(* CODESYS project BatteryPicker.project
   Company: LCP
   DefaultNamespace: LCP_RoboticApplication
   Title: LCP_PnP_Motion_Master
   Version: 1.0

Project tree, tasks and I/O mapping:
  Controller_3200C : Controller 3200C, Lenze, order no. LPC 1000, version 3.13.0.2
    application Application
      libraries: ModbusTCP Slave, * (3S - Smart Software Solutions GmbH); CAA Types, 3.0.0.2 (3S - Smart Software Solutions GmbH); CAA File, * (CAA Technical Workgroup); L_CT1P_ControlToolbox, * (Lenze); L_Util, 3.13.0.0 (Lenze); L_PLCDataManagerAccess, 3.0.0.0 (Lenze); L_PLCLoggingAccess, 3.3.0.0 (Lenze); L_IE1P_ApplicationErrors, 3.13.1.0 (Lenze); L_MC4P_RoboticHandling, 3.13.2.5 (Lenze); L_IODrvEtherCAT, 3.12.0.0 (Lenze); SysTimeCore, * (System); CAA Net Base Services, * (CAA Technical Workgroup); L_USPP_SignalProcessing, * (Lenze); L_MC1P_MotionControlBasic, 3.13.1.0 (Lenze); L_MC2P_MotionControlCam, 3.13.1.56 (Lenze); L_DCO_DriveCommunication, 3.1.0.0 (Lenze); SysMem, * (System); CAA Mathematics, * (CAA Technical Workgroup); LCP_PnP_Ellipse_Motion, 2.0 (LCP); CAA Memory, * (CAA Technical Workgroup)
      task Motion (cyclic, interval t#1ms, priority 1, watchdog t#2ms x 1) calls Main
      task Logic (cyclic, interval t#5ms, priority 2) calls LogicControl
      program Main [ST]: A00_Init, A20_ManualJog, A30_AutoRun, A80_SuckBlow, A60_CameraHandler, A93_SetTorqueLimit, A02_DetectDeviceChoose, A03_PowerCtrl, A04_ResetFunction, A40_SetParameters, A94_RealAxisFilter, A96_IK, A98_TFFControl
      B0_GloabalVariables/
        global variables PersistentVars
        global variables L_MC4P_AGBC_VARS
        global variables GVL_Const
        global variables PrgVars
        global variables GVL_MainFlow
        global variables PPVars
        global variables GVL_HardwareIO
      B1_STRUCT/
        data type sRobotPos
        data type CalibratePt
        data type Detect_Device
        data type Display_Product
      B5_VISUAL/
        visualisation DeltaRobot
        visualisation ABControl
        visualisation Products
        visualisation SensorBuffer
        visualisation MultiPick
      program LogicControl [ST]: A40_Modbus_Slave, A20_StatusDisplay, A10_CameraInterface, A01_EditPrg, A10_Homing, A50_Brake
      B6_TRACE/
        trace RobotStatus (task Motion): CustomerPrgHandling.iAutoStep, Delta_Robot.lrPathVelocity, Delta_Robot.lrPathAcceleration, CustomerPrgHandling.BoxBuffer.NewProd_Rtrig.Q, Infeeder.lrActPosition, Infeeder.lrActVelocity, Infeeder.lrActAcceleration, CustomerPrgHandling.MC_TrackConveyorBelt_U1.Busy, CustomerPrgHandling.MC_TrackConveyorBelt_U1.Active, CustomerPrgHandling.MC_TrackConveyorBelt_U1.InSync, CustomerPrgHandling.MC_TrackConveyorBelt_U1.Done, Outfeeder.lrActPosition, Outfeeder.lrActVelocity, Outfeeder.lrActAcceleration, CustomerPrgHandling.MC_TrackConveyorBelt_U2.Busy, CustomerPrgHandling.MC_TrackConveyorBelt_U2.Active, CustomerPrgHandling.MC_TrackConveyorBelt_U2.InSync, CustomerPrgHandling.MC_TrackConveyorBelt_U2.Done, CustomerPrgHandling.MC_TrackConveyorBelt_U2.Abort, CustomerPrgHandling.MC_TrackConveyorBelt_U2.CommandAborted, CustomerPrgHandling.L_RPP_PickPlace_0.Busy, CustomerPrgHandling.L_RPP_PickPlace_1.Busy, CustomerPrgHandling.L_RPP_PickPlace_1.xBusyTemp, CustomerPrgHandling.L_RPP_PickPlace_1.SWOut, CustomerPrgHandling.MoveToWaitPoint0.Busy, CustomerPrgHandling.MoveToWaitPoint0.Active, CustomerPrgHandling.MoveToWaitPoint0.Done, CustomerPrgHandling.BoxBuffer.xFirstProdDel, CustomerPrgHandling.BoxBuffer.xProdInfoReady, CustomerPrgHandling.BoxBuffer.sFirstProdInfo.lrDeltaX, CustomerPrgHandling.BoxBuffer.lrPosFirstProdInfo, CustomerPrgHandling.BoxBuffer.iNewProdCount, A1.lrActTorque, A2.lrActTorque, A3.lrActTorque, AxisYaw.lrActTorque, A1.lrActFollowingError, A2.lrActFollowingError, A3.lrActFollowingError, AxisYaw.lrActFollowingError
        trace Trace (task Motion): Axis_X.lrSetPosition, Axis_Y.lrSetPosition, Axis_Z.lrSetPosition, Axis_X.lrActPosition, Axis_Y.lrActPosition, Axis_Z.lrActPosition, Axis_X.lrSetAcceleration, Axis_Y.lrSetAcceleration, Axis_Z.lrSetAcceleration, Delta_Robot.lrPathVelocity, Delta_Robot.lrPathAcceleration, A1.lrSetAcceleration, A2.lrSetAcceleration, A3.lrSetAcceleration, A1.lrActPosition, A2.lrActPosition, A3.lrActPosition, A1.lrActTorque, A2.lrActTorque, A3.lrActTorque, A1.lrActFollowingError, A2.lrActFollowingError, A3.lrActFollowingError
        trace RobotPerformance (task Motion): CustomerPrgHandling.L_RPP_PickPlace_0.Busy, CustomerPrgHandling.L_RPP_PickPlace_1.Busy, Axis_X.lrSetPosition, Axis_Y.lrSetPosition, Axis_Z.lrSetPosition, Axis_X.lrActPosition, Axis_Y.lrActPosition, Axis_Z.lrActPosition, Axis_X.lrSetAcceleration, Axis_Y.lrSetAcceleration, Axis_Z.lrSetAcceleration, Delta_Robot.lrPathVelocity, Delta_Robot.lrPathAcceleration, A1.lrActPosition, A2.lrActPosition, A3.lrActPosition, A1.lrActTorque, A2.lrActTorque, A3.lrActTorque, A1.lrActFollowingError, A2.lrActFollowingError, A3.lrActFollowingError
        trace ErrorID (task Motion): DeltaRobot_ErrorID, A1axis_ErrorID, A2axis_ErrorID, A3axis_ErrorID, AuxCaxis_ErrorID, Xaxis_ErrorID, Yaxis_ErrorID, Zaxis_ErrorID, ErrorID, Main.LoadDistribution.xOverlap, Main.LoadDistribution.xProductNew
        trace Trace_1 (task Motion): CustomerPrgHandling.iAutoStep
        trace PathLength_DurationInternal (task Motion): CustomerPrgHandling.L_RPP_PickPlace_0.Ellipse_Cal_Pts.lrPathLength, CustomerPrgHandling.L_RPP_PickPlace_1.Ellipse_Cal_Pts.lrPathLength, CustomerPrgHandling.L_RPP_PickPlace_0.lrDurationInternal, CustomerPrgHandling.L_RPP_PickPlace_1.lrDurationInternal
        trace Trace_2 (task Motion): CustomerPrgHandling.L_RPP_PickPlace_0.Busy, CustomerPrgHandling.L_RPP_PickPlace_1.Busy, Axis_X.lrSetPosition, Axis_Y.lrSetPosition, Axis_Z.lrSetPosition, Axis_X.lrActPosition, Axis_Y.lrActPosition, Axis_Z.lrActPosition, Axis_X.lrSetAcceleration, Axis_Y.lrSetAcceleration, Axis_Z.lrSetAcceleration, Delta_Robot.lrPathVelocity, Delta_Robot.lrPathAcceleration, A1.lrActPosition, A2.lrActPosition, A3.lrActPosition, A1.lrActTorque, A2.lrActTorque, A3.lrActTorque, A1.lrActFollowingError, A2.lrActFollowingError, A3.lrActFollowingError
      program CustomerPrgHandling [ST]: A01_PickAlone, A02_PlaceAlone, A00_ProgramHandling, A03_RobotSateTransition
      FunctionBlock/
        function block FourPts_Calibration [ST]
        function _L_MC1B_PackBytesToDWord [ST]
        function _L_MC1B_PackBytesToLreal [ST]
        function _L_MC1B_PackBytesToWord [ST]
        function _L_MC1B_PackDWordToByte [ST]
        function _L_MC1B_PackLRealToByte [ST]
        function _L_MC1B_PackWordToByte [ST]
      TorqueFeedforwardControl/
        trace Dynamics (task TaskHighPriority): Axis_X.lrSetPosition, Axis_Y.lrSetPosition, Axis_Z.lrSetPosition, Axis_X.lrSetVelocity, Axis_Y.lrSetVelocity, Axis_Z.lrSetVelocity, Axis_X.lrSetAcceleration, Axis_Y.lrSetAcceleration, Axis_Z.lrSetAcceleration, A1.lrSetPosition, A2.lrSetPosition, A3.lrSetPosition, A1.lrSetVelocity, A2.lrSetVelocity, A3.lrSetVelocity, A1.lrSetAcceleration, A2.lrSetAcceleration, A3.lrSetAcceleration, A1.lrActTorque, A2.lrActTorque, A3.lrActTorque, A1.lrActFollowingError, A2.lrActFollowingError, A3.lrActFollowingError
        trace Trace_Theta (task Motion): Main.fb_InverseKinematics.theta1, Main.fb_InverseKinematics.theta2, Main.fb_InverseKinematics.theta3, A1.lrSetPosition, A2.lrSetPosition, A3.lrSetPosition
        trace Trace_Torque (task Motion): CustomerPrgHandling.L_RPP_PickPlace_1.Busy, A1.lrActTorque, A2.lrActTorque, A3.lrActTorque, Axis_X.lrSetPosition, Axis_Y.lrSetPosition, Axis_Z.lrSetPosition, Main.LCP_MC4P_TorqueComputation_1.alrComputedTorque[1], Main.LCP_MC4P_TorqueComputation_1.alrComputedTorque[2], Main.LCP_MC4P_TorqueComputation_1.alrComputedTorque[3], Main.LCP_MC4P_TorqueComputation_1.alrSetTorqueOut[1], Main.LCP_MC4P_TorqueComputation_1.alrSetTorqueOut[2], Main.LCP_MC4P_TorqueComputation_1.alrSetTorqueOut[3], A1.lrSetTorqueToDrive, A2.lrSetTorqueToDrive, A3.lrSetTorqueToDrive, A1.lrActFollowingError, A2.lrActFollowingError, A3.lrActFollowingError
        trace Torque (task Motion): A1.lrActTorque, A2.lrActTorque, A3.lrActTorque, Main.fb_SimplifiedTorqueComputationKorea.tau1, Main.fb_SimplifiedTorqueComputationKorea.tau2, Main.fb_SimplifiedTorqueComputationKorea.tau3, Main.fb_SimplifiedTorqueComputationGermany.tau1, Main.fb_SimplifiedTorqueComputationGermany.tau2, Main.fb_SimplifiedTorqueComputationGermany.tau3, Main.fb_CompleteTorqueComputationSpain.tau1, Main.fb_CompleteTorqueComputationSpain.tau2, Main.fb_CompleteTorqueComputationSpain.tau3, Main.lrAverageTorque[1], Main.lrAverageTorque[2], Main.lrAverageTorque[3], A1.lrActFollowingError, A2.lrActFollowingError, A3.lrActFollowingError, A1.lrSetTorqueToDrive, A2.lrSetTorqueToDrive, A3.lrSetTorqueToDrive
        trace Trace_4 (task Motion): CustomerPrgHandling.L_RPP_PickPlace_0.Busy, A1.lrActTorque, A2.lrActTorque, A3.lrActTorque, Main.fb_SimplifiedTorqueComputation.tau1, Main.fb_SimplifiedTorqueComputation.tau2, Main.fb_SimplifiedTorqueComputation.tau3, Main.fb_SimplifiedTorqueComputation.alrFriction[1], Main.fb_SimplifiedTorqueComputation.alrFriction[2], Main.fb_SimplifiedTorqueComputation.alrFriction[3], A1.lrSetTorqueToDrive, A2.lrSetTorqueToDrive, A3.lrSetTorqueToDrive, A1.lrActFollowingError, A2.lrActFollowingError, A3.lrActFollowingError
        trace Torque_1 (task Motion): CustomerPrgHandling.L_RPP_PickPlace_0.Busy, A1.lrActTorque, A2.lrActTorque, A3.lrActTorque, Main.fb_SimplifiedTorqueComputationGermany.tau1, Main.fb_SimplifiedTorqueComputationGermany.tau2, Main.fb_SimplifiedTorqueComputationGermany.tau3, Main.fb_SimplifiedTorqueComputationGermany.alrFriction[1], Main.fb_SimplifiedTorqueComputationGermany.alrFriction[2], Main.fb_SimplifiedTorqueComputationGermany.alrFriction[3], A1.lrActFollowingError, A2.lrActFollowingError, A3.lrActFollowingError, A1.lrSetTorqueToDrive, A2.lrSetTorqueToDrive, A3.lrSetTorqueToDrive
        trace Trace_5 (task Motion): Main.fb_InverseKinematics.theta1, Main.fb_InverseKinematics.theta2, Main.fb_InverseKinematics.theta3, A1.lrSetPosition, A2.lrSetPosition, A3.lrSetPosition
        trace Trace_6 (task Motion): A1.lrActTorque, A2.lrActTorque, A3.lrActTorque, Main.fb_SimplifiedTorqueComputationKorea.tau1, Main.fb_SimplifiedTorqueComputationKorea.tau2, Main.fb_SimplifiedTorqueComputationKorea.tau3, Main.fb_SimplifiedTorqueComputationGermany.tau1, Main.fb_SimplifiedTorqueComputationGermany.tau2, Main.fb_SimplifiedTorqueComputationGermany.tau3, Main.fb_CompleteTorqueComputationSpain.tau1, Main.fb_CompleteTorqueComputationSpain.tau2, Main.fb_CompleteTorqueComputationSpain.tau3, Main.lrAverageTorque[1], Main.lrAverageTorque[2], Main.lrAverageTorque[3], A1.lrActFollowingError, A2.lrActFollowingError, A3.lrActFollowingError, A1.lrSetTorqueToDrive, A2.lrSetTorqueToDrive, A3.lrSetTorqueToDrive
        trace L_TT1P_TrackPickAndPlace (task TaskHighPriority): Axis_X.lrSetPosition, Axis_Y.lrSetPosition, Axis_Z.lrSetPosition, Axis_X.lrSetVelocity, Axis_Y.lrSetVelocity, Axis_Z.lrSetVelocity, Axis_X.lrSetAcceleration, Axis_Y.lrSetAcceleration, Axis_Z.lrSetAcceleration, A1.lrSetPosition, A2.lrSetPosition, A3.lrSetPosition, A1.lrSetVelocity, A2.lrSetVelocity, A3.lrSetVelocity, A1.lrSetAcceleration, A2.lrSetAcceleration, A3.lrSetAcceleration, A1.lrActTorque, A2.lrActTorque, A3.lrActTorque, A1.lrActFollowingError, A2.lrActFollowingError, A3.lrActFollowingError
        trace LCP_MC4P_MoveBSpline (task Motion): Axis_X.lrSetPosition, Axis_Y.lrSetPosition, Axis_Z.lrSetPosition, Axis_X.lrSetVelocity, Axis_Y.lrSetVelocity, Axis_Z.lrSetVelocity, Axis_X.lrSetAcceleration, Axis_Y.lrSetAcceleration, Axis_Z.lrSetAcceleration, A1.lrSetPosition, A2.lrSetPosition, A3.lrSetPosition, A1.lrSetVelocity, A2.lrSetVelocity, A3.lrSetVelocity, A1.lrSetAcceleration, A2.lrSetAcceleration, A3.lrSetAcceleration, A1.lrActTorque, A2.lrActTorque, A3.lrActTorque, A1.lrActFollowingError, A2.lrActFollowingError, A3.lrActFollowingError
        trace ErrorAnalysis (task ): xSystemWarning, xSystemError, ErrorID, WarningID, Delta_Robot.eActiveErrorID, Axis_X.eActiveErrorID, Axis_Y.eActiveErrorID, Axis_Z.eActiveErrorID, A1.eActiveErrorID, A2.eActiveErrorID, A3.eActiveErrorID
      A10-Structs/
        A11-scCommunication/
          data type scDataMotion_FromPLC
          data type scDataMotion_ToPLC
        A12_scControlWord/
          data type scDataControlWord_1_FromPLC
        A13_scStatusWord/
          data type scDataMotionStatusWord_1_ToPLC
        A14_scPnP_Data/
          data type scPnP_Data
        data type scWord_to_bits
        A15_SlaveStatetoMaster/
          data type eSlaveToMaster_State
      A20-Unions/
        data type scDataMotion_ToSiemens
        data type scDataMotion_FromSiemens
      A30_Enum/
        A31_AutoRunStep/
          data type eAutoRun_Step
    Coupler_I_O_moduls : Coupler I/O moduls, Lenze, version 3.6.0.0
        settings: Count groups = 1; Application Name of Task = 'Application'; Group1 Task Name = 'Motion'
        unmapped channels: Error, unused, unused, unused, unused, unused, unused, unused, ErrorID, AbsoluteCounter, ErrorReset, unused, unused, unused, unused, unused, unused, unused
      EPM_S202 : EPM-S202: DI8, DC 24V, Lenze, order no. EPM-S202, version 3.6.0.0
          settings: Group = 0; Task Guid = '00000000-0000-0000-0000-000000000000'
          unmapped channels: DI1, DI2, DI3, DI4, DI5, DI6, DI7, DI8
      EPM_S302 : EPM-S302: DO8, DC 24V, 0.5A, Lenze, order no. EPM-S302, version 3.6.0.0
          settings: Group = 0; Task Guid = '00000000-0000-0000-0000-000000000000'
          unmapped channels: DO1, DO2, DO3, DO4, DO5, DO6, DO7, DO8
    AxesGroups
      Delta_Robot : Delta3_3dof, Lenze, version 3.9.0.0
          settings: BaseIndex = 20992 AXIS_REF.BaseIndex.Unit
        Axis_X : LM_Virtual_Drive, Lenze, version 3.9.0.0
            settings: BaseIndex = 20736 AXIS_REF.BaseIndex.Unit
        Axis_Y : LM_Virtual_Drive, Lenze, version 3.9.0.0
            settings: BaseIndex = 20737 AXIS_REF.BaseIndex.Unit
        Axis_Z : LM_Virtual_Drive, Lenze, version 3.9.0.0
            settings: BaseIndex = 20738 AXIS_REF.BaseIndex.Unit
    VirtualAxes
      AxisYaw : LM_Virtual_Drive, Lenze, version 3.9.0.0
          settings: BaseIndex = 20774 AXIS_REF.BaseIndex.Unit; Guid1 = 4273197094; Guid2 = 1328921582; Guid3 = 3991759762; Guid4 = 3302118515
      Outfeeder : LM_Virtual_Drive, Lenze, version 3.9.0.0
          settings: BaseIndex = 20768 AXIS_REF.BaseIndex.Unit; Guid1 = 443594626; Guid2 = 1335482620; Guid3 = 2315861686; Guid4 = 2195944928
      Infeeder : LM_Virtual_Drive, Lenze, version 3.9.0.0
          settings: BaseIndex = 20767 AXIS_REF.BaseIndex.Unit; Guid1 = 1238477134; Guid2 = 1229563840; Guid3 = 1829875085; Guid4 = 3937990101
    EtherCAT_Master : EtherCAT Master, Lenze, version 3.12.0.1
        settings: MasterCycleTime = 1000; TimeoutInitToPreOP = 3000; TimeoutPreOpToSafeOpToOp = 10000
      L_i700 : i700 (Single Inverter, Safety STO) FW V01.10, Lenze, version 1.10.12.0
          settings: DC sync0 cycletime = 1000; DC sync1 cycletime = 1000
          unmapped channels: Controlword, Lenze control word, Modes of operation, Torque offset, Target position, Velocity offset, Speed controller: I component load value, Touch probe function, Positive torque limit value, Negative torque limit value, Speed limitation: Upper speed limit, Speed limitation: Lower speed limit, Statusword, Lenze status word, Modes of operation display, Error code, Velocity actual value, Torque actual value, Position actual value, Following error actual value, Touch probe status, Touch probe pos1 pos value, Touch probe pos1 neg value, Touch probe pos2 pos value, Touch probe pos2 neg value, Lenze statusword 2, Digital inputs
        A1 : i700_ETC_Motion_Axis, Lenze, version 3.12.0.0
            settings: BaseIndex = 20771 AXIS_REF.BaseIndex.Unit; Controlword = '%QW2'; Controlword = '16'; Controlword = ADR(%QW2); Controlword = 16; ModesOfOperation = '%QB8'; ModesOfOperation = '8'; ModesOfOperation = ADR(%QB8); ModesOfOperation = 8; TargetPosition = '%QD3'; TargetPosition = '32'; TargetPosition = ADR(%QD3); TargetPosition = 32; TorqueLimitPos = '%QW12'; TorqueLimitPos = '16'; TorqueLimitPos = ADR(%QW12); TorqueLimitPos = 16; TorqueLimitNeg = '%QW13'; TorqueLimitNeg = '16'; TorqueLimitNeg = ADR(%QW13); TorqueLimitNeg = 16; SpeedLimHigh = '%QD7'; SpeedLimHigh = '32'; SpeedLimHigh = ADR(%QD7); SpeedLimHigh = 32; SpeedLimLow = '%QD8'; SpeedLimLow = '32'; SpeedLimLow = ADR(%QD8); SpeedLimLow = 32; TPControl = '%QW11'; TPControl = '16'; TPControl = ADR(%QW11); TPControl = 16; OffsetVelocity = '%QD4'; OffsetVelocity = '32'; OffsetVelocity = ADR(%QD4); OffsetVelocity = 32; OffsetTorque = '%QW5'; OffsetTorque = '16'; OffsetTorque = ADR(%QW5);
              OffsetTorque = 16; SpeedCtrlLoad = '%QW10'; SpeedCtrlLoad = '16'; SpeedCtrlLoad = ADR(%QW10); SpeedCtrlLoad = 16; LenzeCtrl = '%QW3'; LenzeCtrl = '16'; LenzeCtrl = ADR(%QW3); LenzeCtrl = 16; Statusword = '%IW6'; Statusword = '16'; Statusword = ADR(%IW6); Statusword = 16; ModesOfOperationDisplay = '%IB16'; ModesOfOperationDisplay = '8'; ModesOfOperationDisplay = ADR(%IB16); ModesOfOperationDisplay = 8; ActualPosition = '%ID7'; ActualPosition = '32'; ActualPosition = ADR(%ID7); ActualPosition = 32; ActualVelocity = '%ID5'; ActualVelocity = '32'; ActualVelocity = ADR(%ID5); ActualVelocity = 32; ActualTorque = '%IW12'; ActualTorque = '16'; ActualTorque = ADR(%IW12); ActualTorque = 16; ErrorCode = '%IW9'; ErrorCode = '16'; ErrorCode = ADR(%IW9); ErrorCode = 16; FollowingError = '%ID8'; FollowingError = '32'; FollowingError = ADR(%ID8); FollowingError = 32; LenzeState = '%IW7'; LenzeState = '16'; LenzeState = ADR(%IW7);
              LenzeState = 16; LenzeState2 = '%IW28'; LenzeState2 = '16'; LenzeState2 = ADR(%IW28); LenzeState2 = 16; TPState = '%IW18'; TPState = '16'; TPState = ADR(%IW18); TPState = 16; TP1Pos = '%ID10'; TP1Pos = '32'; TP1Pos = ADR(%ID10); TP1Pos = 32; TP1Neg = '%ID11'; TP1Neg = '32'; TP1Neg = ADR(%ID11); TP1Neg = 32; TP2Pos = '%ID12'; TP2Pos = '32'; TP2Pos = ADR(%ID12); TP2Pos = 32; TP2Neg = '%ID13'; TP2Neg = '32'; TP2Neg = ADR(%ID13); TP2Neg = 32; DigitalInputs = '%ID15'; DigitalInputs = '32'; DigitalInputs = ADR(%ID15); DigitalInputs = 32; Guid1 = 4196502328; Guid2 = 1146177473; Guid3 = 2028349326; Guid4 = 3167738062
      L_i700_1 : i700 (Double Inverter, Safety STO) FW V01.10, Lenze, version 1.10.12.0
          settings: DC sync0 cycletime = 1000; DC sync1 cycletime = 1000
          unmapped channels: Controlword, Lenze control word, Modes of operation, Torque offset, Target position, Velocity offset, Speed controller: I component load value, Touch probe function, Positive torque limit value, Negative torque limit value, Speed limitation: Upper speed limit, Speed limitation: Lower speed limit, Controlword, Lenze control word, Modes of operation, Torque offset, Target position, Velocity offset, Speed controller: I component load value, Touch probe function, Positive torque limit value, Negative torque limit value, Speed limitation: Upper speed limit, Speed limitation: Lower speed limit, Statusword, Lenze status word, Modes of operation display, Error code, Velocity actual value, Torque actual value, Position actual value, Following error actual value, Touch probe status, Touch probe pos1 pos value, Touch probe pos1 neg value, Touch probe pos2 pos value, Touch probe pos2 neg value, Lenze statusword 2, Digital inputs, Statusword,
            Lenze status word, Modes of operation display, Error code, Velocity actual value, Torque actual value, Position actual value, Following error actual value, Touch probe status, Touch probe pos1 pos value, Touch probe pos1 neg value, Touch probe pos2 pos value, Touch probe pos2 neg value, Lenze statusword 2, Digital inputs
        A2 : i700_ETC_Motion_Axis, Lenze, version 3.12.0.0
            settings: BaseIndex = 20772 AXIS_REF.BaseIndex.Unit; Controlword = '%QW18'; Controlword = '16'; Controlword = ADR(%QW18); Controlword = 16; ModesOfOperation = '%QB40'; ModesOfOperation = '8'; ModesOfOperation = ADR(%QB40); ModesOfOperation = 8; TargetPosition = '%QD11'; TargetPosition = '32'; TargetPosition = ADR(%QD11); TargetPosition = 32; TorqueLimitPos = '%QW28'; TorqueLimitPos = '16'; TorqueLimitPos = ADR(%QW28); TorqueLimitPos = 16; TorqueLimitNeg = '%QW29'; TorqueLimitNeg = '16'; TorqueLimitNeg = ADR(%QW29); TorqueLimitNeg = 16; SpeedLimHigh = '%QD15'; SpeedLimHigh = '32'; SpeedLimHigh = ADR(%QD15); SpeedLimHigh = 32; SpeedLimLow = '%QD16'; SpeedLimLow = '32'; SpeedLimLow = ADR(%QD16); SpeedLimLow = 32; TPControl = '%QW27'; TPControl = '16'; TPControl = ADR(%QW27); TPControl = 16; OffsetVelocity = '%QD12'; OffsetVelocity = '32'; OffsetVelocity = ADR(%QD12); OffsetVelocity = 32; OffsetTorque = '%QW21'; OffsetTorque = '16'; OffsetTorque = ADR(%QW21);
              OffsetTorque = 16; SpeedCtrlLoad = '%QW26'; SpeedCtrlLoad = '16'; SpeedCtrlLoad = ADR(%QW26); SpeedCtrlLoad = 16; LenzeCtrl = '%QW19'; LenzeCtrl = '16'; LenzeCtrl = ADR(%QW19); LenzeCtrl = 16; Statusword = '%IW32'; Statusword = '16'; Statusword = ADR(%IW32); Statusword = 16; ModesOfOperationDisplay = '%IB68'; ModesOfOperationDisplay = '8'; ModesOfOperationDisplay = ADR(%IB68); ModesOfOperationDisplay = 8; ActualPosition = '%ID20'; ActualPosition = '32'; ActualPosition = ADR(%ID20); ActualPosition = 32; ActualVelocity = '%ID18'; ActualVelocity = '32'; ActualVelocity = ADR(%ID18); ActualVelocity = 32; ActualTorque = '%IW38'; ActualTorque = '16'; ActualTorque = ADR(%IW38); ActualTorque = 16; ErrorCode = '%IW35'; ErrorCode = '16'; ErrorCode = ADR(%IW35); ErrorCode = 16; FollowingError = '%ID21'; FollowingError = '32'; FollowingError = ADR(%ID21); FollowingError = 32; LenzeState = '%IW33'; LenzeState = '16'; LenzeState = ADR(%IW33);
              LenzeState = 16; LenzeState2 = '%IW54'; LenzeState2 = '16'; LenzeState2 = ADR(%IW54); LenzeState2 = 16; TPState = '%IW44'; TPState = '16'; TPState = ADR(%IW44); TPState = 16; TP1Pos = '%ID23'; TP1Pos = '32'; TP1Pos = ADR(%ID23); TP1Pos = 32; TP1Neg = '%ID24'; TP1Neg = '32'; TP1Neg = ADR(%ID24); TP1Neg = 32; TP2Pos = '%ID25'; TP2Pos = '32'; TP2Pos = ADR(%ID25); TP2Pos = 32; TP2Neg = '%ID26'; TP2Neg = '32'; TP2Neg = ADR(%ID26); TP2Neg = 32; DigitalInputs = '%ID28'; DigitalInputs = '32'; DigitalInputs = ADR(%ID28); DigitalInputs = 32; Guid1 = 1181001955; Guid2 = 1284246117; Guid3 = 3320666543; Guid4 = 734373032
        A3 : i700_ETC_Motion_Axis_B, Lenze, version 3.12.0.0
            settings: BaseIndex = 20773 AXIS_REF.BaseIndex.Unit; Controlword = '%QW34'; Controlword = '16'; Controlword = ADR(%QW34); Controlword = 16; ModesOfOperation = '%QB72'; ModesOfOperation = '8'; ModesOfOperation = ADR(%QB72); ModesOfOperation = 8; TargetPosition = '%QD19'; TargetPosition = '32'; TargetPosition = ADR(%QD19); TargetPosition = 32; TorqueLimitPos = '%QW44'; TorqueLimitPos = '16'; TorqueLimitPos = ADR(%QW44); TorqueLimitPos = 16; TorqueLimitNeg = '%QW45'; TorqueLimitNeg = '16'; TorqueLimitNeg = ADR(%QW45); TorqueLimitNeg = 16; SpeedLimHigh = '%QD23'; SpeedLimHigh = '32'; SpeedLimHigh = ADR(%QD23); SpeedLimHigh = 32; SpeedLimLow = '%QD24'; SpeedLimLow = '32'; SpeedLimLow = ADR(%QD24); SpeedLimLow = 32; TPControl = '%QW43'; TPControl = '16'; TPControl = ADR(%QW43); TPControl = 16; OffsetVelocity = '%QD20'; OffsetVelocity = '32'; OffsetVelocity = ADR(%QD20); OffsetVelocity = 32; OffsetTorque = '%QW37'; OffsetTorque = '16'; OffsetTorque = ADR(%QW37);
              OffsetTorque = 16; SpeedCtrlLoad = '%QW42'; SpeedCtrlLoad = '16'; SpeedCtrlLoad = ADR(%QW42); SpeedCtrlLoad = 16; LenzeCtrl = '%QW35'; LenzeCtrl = '16'; LenzeCtrl = ADR(%QW35); LenzeCtrl = 16; Statusword = '%IW58'; Statusword = '16'; Statusword = ADR(%IW58); Statusword = 16; ModesOfOperationDisplay = '%IB120'; ModesOfOperationDisplay = '8'; ModesOfOperationDisplay = ADR(%IB120); ModesOfOperationDisplay = 8; ActualPosition = '%ID33'; ActualPosition = '32'; ActualPosition = ADR(%ID33); ActualPosition = 32; ActualVelocity = '%ID31'; ActualVelocity = '32'; ActualVelocity = ADR(%ID31); ActualVelocity = 32; ActualTorque = '%IW64'; ActualTorque = '16'; ActualTorque = ADR(%IW64); ActualTorque = 16; ErrorCode = '%IW61'; ErrorCode = '16'; ErrorCode = ADR(%IW61); ErrorCode = 16; FollowingError = '%ID34'; FollowingError = '32'; FollowingError = ADR(%ID34); FollowingError = 32; LenzeState = '%IW59'; LenzeState = '16'; LenzeState = ADR(%IW59);
              LenzeState = 16; LenzeState2 = '%IW80'; LenzeState2 = '16'; LenzeState2 = ADR(%IW80); LenzeState2 = 16; TPState = '%IW70'; TPState = '16'; TPState = ADR(%IW70); TPState = 16; TP1Pos = '%ID36'; TP1Pos = '32'; TP1Pos = ADR(%ID36); TP1Pos = 32; TP1Neg = '%ID37'; TP1Neg = '32'; TP1Neg = ADR(%ID37); TP1Neg = 32; TP2Pos = '%ID38'; TP2Pos = '32'; TP2Pos = ADR(%ID38); TP2Pos = 32; TP2Neg = '%ID39'; TP2Neg = '32'; TP2Neg = ADR(%ID39); TP2Neg = 32; DigitalInputs = '%ID41'; DigitalInputs = '32'; DigitalInputs = ADR(%ID41); DigitalInputs = 32; Guid1 = 1028340755; Guid2 = 1121766493; Guid3 = 837655470; Guid4 = 3735374898
    PROFINET_Device : PROFINET Device, Lenze, version 3.14.0.0
        settings: Io Device Identification.IP address = [192,168,2,60]; Io Device Identification.Default gateway = [192,168,2,1]; Io Device Identification.Station name = 'ROB-NG2'
      Slave_Out_Master_In_Word_0016 : Slave-Out / Master-In Word 0016, Lenze, version 3.14.0.0
          output Application.CustomerPrgHandling.scDataInformation_ToSiemens : TWordArray16  // Out
      Slave_In_Master_Out_Word_0256 : Slave-In / Master-Out Word 0256, Lenze, version 3.14.0.0
          settings: Io Device Submodule.Slot number = 3
          input  Application.CustomerPrgHandling.scDataInformation_FromSiemens.scDataMotionFromPLC.aPalletInformation : TWordArray256  // In
      Slave_In_Master_Out_Byte_0004 : Slave-In / Master-Out Byte 0004, Lenze, version 3.14.0.0
          settings: Io Device Submodule.Slot number = 2
          input  Application.CustomerPrgHandling.scDataInformation_FromSiemens.scDataMotionFromPLC.wCtrl_2 : TByteArray4  // In
  text list GlobalTextList
*)

// Controller_3200C/Application/B1_STRUCT/sRobotPos
TYPE sRobotPos :
STRUCT
	rRobotPosX			:REAL;
	rRobotPosY			:REAL;
	rRobotPosZ			:REAL;
	rRobotPosC			:REAL;
	rRobotPosA1		    :REAL;
	rRobotPosA2		    :REAL;
	rRobotPosA3		    :REAL;
END_STRUCT
END_TYPE

// Controller_3200C/Application/B1_STRUCT/CalibratePt
TYPE CalibratePt :
STRUCT
	rX: REAL;
    rY: REAL;
    rZ: REAL;
END_STRUCT
END_TYPE

// Controller_3200C/Application/B1_STRUCT/Detect_Device
{attribute 'strict'}
TYPE Detect_Device :
(
	Camera := 0,
	Sensor := 1,
	Computer:=2
);
END_TYPE

// Controller_3200C/Application/B1_STRUCT/Display_Product
TYPE Display_Product :
STRUCT
	iAttribute				: INT; 		//  属性				
	lrCameraPosX			: REAL;	//	拍照时X坐标				
	lrCameraPosY			: REAL;	//	拍照时y坐标		
	lrCameraPosAuxC			: REAL;	//	拍照时c坐标 
END_STRUCT
END_TYPE

// Controller_3200C/Application/A10-Structs/A11-scCommunication/scDataMotion_FromPLC
TYPE scDataMotion_FromPLC :
STRUCT
	wCtrl_2							:scDataControlWord_1_FromPLC;	// 4个byte=2个word=32个bit
	aPalletInformation				:ARRAY[1..256] OF WORD;	//上位机传来的码盘信息	0 为不抓，非0为抓,非零索引号代表抓取位置，非零数值代表放置位置			
END_STRUCT
END_TYPE

// Controller_3200C/Application/A10-Structs/A11-scCommunication/scDataMotion_ToPLC
TYPE scDataMotion_ToPLC :
STRUCT
	wCtrl_16						:					scDataMotionStatusWord_1_ToPLC;			// StatusWord 1	
END_STRUCT
END_TYPE

// Controller_3200C/Application/A10-Structs/A12_scControlWord/scDataControlWord_1_FromPLC
TYPE scDataControlWord_1_FromPLC :
STRUCT
	wCtrl_scWord_to_bits1			:					scWord_to_bits;									// 
	wCtrl_scWord_to_bits2			:					scWord_to_bits;									// 
END_STRUCT
END_TYPE

// Controller_3200C/Application/A10-Structs/A13_scStatusWord/scDataMotionStatusWord_1_ToPLC
TYPE scDataMotionStatusWord_1_ToPLC :
STRUCT
	wCtrl_scWord_to_bits1			:					scWord_to_bits;									// 
	wCtrl_scWord_to_bits2			:					scWord_to_bits;									// 
	wCtrl_scWord_to_bits3			:					scWord_to_bits;									// 
	wCtrl_scWord_to_bits4			:					scWord_to_bits;									// 
	wCtrl_scWord_to_bits5			:					scWord_to_bits;									// 
	wCtrl_scWord_to_bits6			:					scWord_to_bits;									// 
	wCtrl_scWord_to_bits7			:					scWord_to_bits;									// 
	wCtrl_scWord_to_bits8			:					scWord_to_bits;									// 
	wCtrl_scWord_to_bits9			:					scWord_to_bits;									// 
	wCtrl_scWord_to_bits10			:					scWord_to_bits;									// 
	wCtrl_scWord_to_bits11			:					scWord_to_bits;									// 
	wCtrl_scWord_to_bits12			:					scWord_to_bits;									// 
	wCtrl_scWord_to_bits13			:					scWord_to_bits;									// 
	wCtrl_scWord_to_bits14			:					scWord_to_bits;									// 
	wCtrl_scWord_to_bits15			:					scWord_to_bits;									// 
	wCtrl_scWord_to_bits16			:					scWord_to_bits;									// 
END_STRUCT
END_TYPE

// Controller_3200C/Application/A10-Structs/A14_scPnP_Data/scPnP_Data
TYPE scPnP_Data :
STRUCT
	xStatus			:BOOL;
	iPickPosition	:INT;
	iPlacePosition	:INT;
END_STRUCT
END_TYPE

// Controller_3200C/Application/A20-Unions/scDataMotion_ToSiemens
TYPE scDataMotion_ToSiemens :
UNION
	aWordDataMotionToPLC			:					ARRAY [1..16] OF WORD;
	scDataMotionToPLC				:					scDataMotion_ToPLC;
END_UNION
END_TYPE

// Controller_3200C/Application/A20-Unions/scDataMotion_FromSiemens
TYPE scDataMotion_FromSiemens :
UNION
	aWordDataMotionFromPLC			:					ARRAY [1..258] OF WORD;//2+256
	scDataMotionFromPLC				:					scDataMotion_FromPLC;
END_UNION
END_TYPE

// Controller_3200C/Application/A10-Structs/scWord_to_bits
TYPE scWord_to_bits :
STRUCT
	xbit1		:					BIT;									// 
	xbit2		:					BIT;									// 
	xbit3		:					BIT;									// 
	xbit4		:					BIT;									// 
	xbit5		:					BIT;									// 
	xbit6		:					BIT;									// 
	xbit7		:					BIT;									// 
	xbit8		:					BIT;									// 
	xbit9		:					BIT;									// 
	xbit10		:					BIT;									// 
	xbit11		:					BIT;									// 
	xbit12		:					BIT;									// 
	xbit13		:					BIT;									// 	
	xbit14		:					BIT;									// 
	xbit15		:					BIT;									// 
	xbit16		:					BIT;									// 	
END_STRUCT
END_TYPE

// Controller_3200C/Application/A10-Structs/A15_SlaveStatetoMaster/eSlaveToMaster_State
{attribute 'strict'}
TYPE eSlaveToMaster_State :
(
	Manual:= 0,
	Waiting,
	Running,
	MotionCompleted,
	Error
);
END_TYPE

// Controller_3200C/Application/A30_Enum/A31_AutoRunStep/eAutoRun_Step
{attribute 'strict'}
TYPE eAutoRun_Step :
(
	NULL := 0,
	P2P_Step,
	MoveLinear_Step,
	MoveCircle_Step,
	Pick_Step,
	Place_Step,
	MoveWaitPoint_Step,
	WaitEvent_Step,
	WaitTime_Step,
	Jump_Step,
	Output_Step
);
END_TYPE

// Controller_3200C/Application/B0_GloabalVariables/PersistentVars
VAR_GLOBAL PERSISTENT RETAIN
	//进料带参数
	p_rConveyorInRecord0					:REAL;
	p_rConveyorInRecord1  					:REAL;
	p_rConveyorInRecord2					:REAL;
	                                		
	p_rReadInfeedPos1_X		    			:REAL;
	p_rReadInfeedPos1_Y		    			:REAL;
	p_rReadInfeedPos1_Z		    			:REAL;
	                                		
	p_rReadInfeedPos2_X		    			:REAL;
	p_rReadInfeedPos2_Y		    			:REAL;
	p_rReadInfeedPos2_Z		    			:REAL;
	                                		
	p_rReadInfeedPos3_X		    			:REAL;
	p_rReadInfeedPos3_Y		    			:REAL;
	p_rReadInfeedPos3_Z		    			:REAL;
	                                		
	p_rReadInfeedPos4_X		    			:REAL;
	p_rReadInfeedPos4_Y		    			:REAL;
	p_rReadInfeedPos4_Z		    			:REAL;
	                                		
	p_theta1								:REAL;
	p_alpha									:REAL;
	p_rInfeedMapX							:REAL;
	p_rInfeedMapY							:REAL;
	
	//出料带参数                             	
	p_rConveyorOutRecord0		 			:REAL;
	p_rConveyorOutRecord1  					:REAL;
	p_rConveyorOutRecord2		  			:REAL;
	                                    	    
	p_rReadOutfeedPos1_X					:REAL;
	p_rReadOutfeedPos1_Y					:REAL;
	p_rReadOutfeedPos1_Z					:REAL;
	                            			    
	p_rReadOutfeedPos2_X					:REAL;
	p_rReadOutfeedPos2_Y					:REAL;
	p_rReadOutfeedPos2_Z					:REAL;
	                                    	
	p_rReadOutfeedPos3_X		    		:REAL;
	p_rReadOutfeedPos3_Y		    		:REAL;
	p_rReadOutfeedPos3_Z		    		:REAL;
	                                    	
	p_rReadOutfeedPos4_X		    		:REAL;
	p_rReadOutfeedPos4_Y		    		:REAL;
	p_rReadOutfeedPos4_Z		    		:REAL;
                                        	
	p_theta2								:REAL;
	p_gama									:REAL;
	
	//PCS5标定 
	p_PCS5_OriginX							:REAL; //坐标系原点 
	p_PCS5_OriginY							:REAL; 
	p_PCS5_OriginZ							:REAL; 
	p_PCS5_OriginA							:REAL; 
	p_PCS5_OriginB							:REAL; 
	p_PCS5_OriginC		 					:REAL; 
	p_PCS5_OriginCRad	     				:REAL; 
	p_PCS5_PX								:REAL; //坐标系X+轴某点 
	p_PCS5_PY								:REAL; 
	p_PCS5_PZ								:REAL; 
                                             
	//PCS6标定                                 
	p_PCS6_OriginX							:REAL; //坐标系原点 
	p_PCS6_OriginY							:REAL; 
	p_PCS6_OriginZ							:REAL; 
	p_PCS6_OriginA							:REAL; 
	p_PCS6_OriginB							:REAL; 
	p_PCS6_OriginC		 					:REAL; 
	p_PCS6_OriginCRad						:REAL; 
	p_PCS6_PX								:REAL; //坐标系X+轴某点 
	p_PCS6_PY								:REAL; 
	p_PCS6_PZ								:REAL; 
	
	p_sInFeedBeltOrigin						:BeltOrigin;  	//以上为计算进料带原点及坐标系所用数据		//1831	
	p_sOutFeedBeltOrigin	 				:BeltOrigin;	//以上为计算出料带原点及坐标系所用数据		//1891
	
	p_PCS5_X0				 				:REAL;
	p_PCS5_Y0                				:REAL;
	p_PCS5_X1                				:REAL;
	p_PCS5_Y1                				:REAL;
	p_PCS5_X2                				:REAL;
	p_PCS5_Y2                				:REAL;
	p_PCS5_X3                				:REAL;
	p_PCS5_Y3                				:REAL;
	p_PCS5_dx                				:REAL;
	p_PCS5_dy                				:REAL;
	                         				
	p_PCS6_X0				 				:REAL;
	p_PCS6_Y0                				:REAL;
	p_PCS6_X1                				:REAL;
	p_PCS6_Y1                				:REAL;
	p_PCS6_X2                				:REAL;
	p_PCS6_Y2                				:REAL;
	p_PCS6_X3                				:REAL;
	p_PCS6_Y3                				:REAL;
	p_PCS6_dx                				:REAL;
	p_PCS6_dy                				:REAL;
	
	p_RobotCalPt1							:CalibratePt;	//1837
	p_RobotCalPt2							:CalibratePt;	//1843
	p_RobotCalPt3							:CalibratePt;	//1849
	p_RobotCalPt4							:CalibratePt;	//1855
	
	p_CameraCalPt1				 			:CalibratePt;	//1861
	p_CameraCalPt2				 			:CalibratePt;	//1867
	p_CameraCalPt3				 			:CalibratePt;	//1873
	p_CameraCalPt4				 			:CalibratePt;	//1879
	
	//自动运行前的相机参数设置
	p_iSuckerNum							:INT;
	p_iCalibSucker							:INT;
	p_rSuker1BiasX				        	:REAL;
	p_rSuker1BiasY				        	:REAL;
	p_rSuker2BiasX				        	:REAL;
	p_rSuker2BiasY				        	:REAL;
	p_rSuker3BiasX				        	:REAL;
	p_rSuker3BiasY				        	:REAL;
	p_rSuker4BiasX				        	:REAL;
	p_rSuker4BiasY				        	:REAL;
	p_rCalibCaxisAngle						:REAL;	
	p_axSavePrgNo							:ARRAY[0..3] OF BOOL;
	p_iCurrentPrgNum						:INT;
	
	//A1轴参数设置                           	
	p_rA1_PositiveLimit			 			:REAL:=20;    
	p_rA1_NegativeLimit			 			:REAL:=-90;   
	p_rA1_Vel_P1		 		 			:REAL:=0.02;
	p_rA1_Vel_I1				 			:REAL:=12;     
	p_rA1_Pos_P1				 			:REAL:=12;    
	//A2轴参数设置
	p_rA2_PositiveLimit						:REAL:=20;    
	p_rA2_NegativeLimit						:REAL:=-90;   
	p_rA2_Vel_P2		 					:REAL:=0.02;
	p_rA2_Vel_I2							:REAL:=12;     
	p_rA2_Pos_P2							:REAL:=12;    
	//A3轴参数设置                           	
	p_rA3_PositiveLimit			 			:REAL:=20;    
	p_rA3_NegativeLimit			 			:REAL:=-90;   
	p_rA3_Vel_P3				 			:REAL:=0.02;
	p_rA3_Vel_I3				 			:REAL:=12;     
	p_rA3_Pos_P3				 			:REAL:=12;    
	//AuxC轴参数设置1                 			
	p_rAuxC_PositiveLimit		 			:REAL:=190;   
	p_rAuxC_NegativeLimit		 			:REAL:=-190;  
	p_rAuxC_Vel_P3				 			:REAL:=0.0175;
	p_rAuxC_Vel_I3				 			:REAL:=8;     
	p_rAuxC_Pos_P3				 			:REAL:=50;       
	//X轴参数设置                     			
	p_rXaxis_PositiveLimit		 			:REAL:=500; 
	p_rXaxis_NegativeLimit		 			:REAL:=-500;
	                        	 			
	//Y轴参数设置                	 			
	p_rYaxis_PositiveLimit		 			:REAL:=400; 
	p_rYaxis_NegativeLimit		 			:REAL:=-450;
	                        	 		
	//Z轴参数设置                	 		
	p_rZaxis_PositiveLimit		 			:REAL:=-700;  
	p_rZaxis_NegativeLimit		 			:REAL:=-915; 
	                                    	
	//Infeeder参数设置                      	
	p_xInfeederDirection					:BOOL:=1;		//方向              
	p_rInfeederPosResolution				:REAL:=2048;	//每圈线数         
	p_rInfeederGearRedRatio					:REAL:=1;		//减速比        
	p_rInfeederFeedConst					:REAL:=200;		//每圈皮带行进长度
	//p_rInfeederCycleLength				:REAL:=10736.8645;	//皮带长度
	
	//Outfeeder参数设置
	p_xOutfeederDirection					:BOOL:=1;		//方向            
	p_rOutfeederPosResolution				:REAL:=1024;  	//每圈线数      
	p_rOutfeederGearRedRatio				:REAL:=1;  		//减速比     
	p_rOutfeederFeedConst					:REAL:=17.6714;  //每圈皮带行进长度
	//p_rOutfeederCycleLength				:REAL:=3733.7885;  //皮带长度
                                        	
	p_i_Suck1_Num							:INT:=5;  	//吸气1 DO端口号
	p_i_Blow1_Num							:INT:=6;  	//吹气1 DO端口号
	//p_iDoShootOut_Num						:INT:=6; 	//相机触发开关 DO端口号
	//p_iPrgDoOutputVal_Num					:INT:=7;  	//程序输出开关 DO端口号
	p_rBoxLength							:REAL;
	p_rBoxBiasLength						:REAL;
	p_iNewProdNum							:INT:=1;
	p_iPrdtDetectDevice						:INT:=0;
	p_rSensorBeltPos						:REAL:=-623;
	p_iBoxTotalPrdoNr						:INT:=72;
	p_rSensorAuxC							:REAL;
	p_rBoxOutfeederVel						:REAL;
	p_rBoxPickTime							:REAL:=0.5;
	p_rBoxPlaceTime							:REAL:=0.5;
	p_rBoxDetectPosX						:REAL;
	                            		
	// 负荷分配                     		
	p_iLoadMode								:INT;
	p_iRobotNum								:INT;
	p_iLoadProdNum							:INT;
	p_iLoadDistrRule						:INT;
	p_arLoadRatio							:ARRAY[1..6] OF REAL; 
	p_aiServerCommuPort						:ARRAY[1..6] OF UINT;
	p_iSlaveCommuPort						:UINT;
	p_xLocal_or_Remote						:BOOL;	
	p_rPallet_DeltaX						:REAL;
	p_rPallet_DeltaY						:REAL;
	p_rPnPDurationNegativeLimit 				:REAL:=0.3;	//13
	P_rPnPDurationPositiveLimit 				:REAL:=0.6;	//14
	p_rTorqueForwardControl						:REAL:=0.7;
	
	p_xExternalMode							:BOOL:=TRUE;
END_VAR

// Controller_3200C/Application/B0_GloabalVariables/L_MC4P_AGBC_VARS
VAR_GLOBAL
	scHomeParamA1A2A3  : L_MC1P_HomeParameter:=(dwTPConfig :=0,
							eHomeMode:= L_MC1P_HomeMode.SetPositionDirect,
							eHomeStopMode:= L_MC1P_HomeStopMode.AbsolutePositioning,
							lrTargetPosition:=0.0,
							lrVelocity1:=5,
							lrVelocity2:=1,
							lrAcceleration1:=50,
							lrAcceleration2:=10,
							lrJerk := 100,
							rTorqueLimit:= 10,
							rTorqueTime:=1,
							wDriveHomeMode:=0);
	lrA1Position		: LREAL :=22.57;
	lrA2Position		: LREAL :=22.57;
	lrA3Position		: LREAL :=22.57;
	ascHomeParam 		: ARRAY[1..12] OF L_MC1P_HomeParameter 	:= [scHomeParamA1A2A3	, scHomeParamA1A2A3	, scHomeParamA1A2A3	];
	alrHomingPosition 	: ARRAY[1..12] OF LREAL;  
	aeHomingOrder		: ARRAY[1..12] OF L_MC4P_HomingOrder	:= [L_MC4P_HomingOrder.FIRST, L_MC4P_HomingOrder.FIRST, L_MC4P_HomingOrder.FIRST]; 
	scParManual			: L_MC4P_AGBC_Parameter := (
							lrCartesianJogVel:= 10, 
							lrCartesianJogAcc:= 100, 
							lrCartesianJogDec:= 200, 
							lrCartesianJogJerk:= 10000, 
							lrOrientationJogVel:= 10, 
							lrOrientationJogAcc:= 50, 
							lrOrientationJogDec:= 100, 
							lrOrientationJogJerk:= 5000, 
							lrRealAxisJogVel:= 10, 
							lrRealAxisJogAcc:= 50, 
							lrRealAxisJogDec:= 100, 
							lrRealAxisJogJerk:= 5000, 
							lrCartesianMoveVel:= 10, 
							lrCartesianMoveAcc:= 100, 
							lrCartesianMoveDec:= 200, 
							lrCartesianMoveJerk:= 10000, 
							lrOrientationMoveVel:= 5, 
							lrOrientationMoveAcc:= 50, 
							lrOrientationMoveDec:= 100, 
							lrOrientationMoveJerk:= 5000, 
							lrRealAxisMoveVel:= 5, 
							lrRealAxisMoveAcc:= 50, 
							lrRealAxisMoveDec:= 100, 
							lrRealAxisMoveJerk:= 5000, 
							lrPathVel:= 50, 
							lrPathAcc:= 100, 
							lrPathDec:= 100, 
							lrPathJerk:= 10000, 
							lrPathStopDec:= 500, 
							lrPathStopJerk:= 50000 , 
							xGroupSetPosRelative:= FALSE, 										
							aeHomingOrder:= aeHomingOrder, 
							xUseHomeExtParameter:= TRUE, 
							ascHomeExtParameter:= ascHomeParam, 
							lrORFadingTime:= 2.5);													
	alrSetPosDist		: ARRAY [1..12] OF LREAL:=[1,1,1,1,1,1];	
	AGBControl			: L_MC4P_AxesGroupBasicControl; //手动控制轴组	 
	Aux1_ABC			: L_MC1P_AxisBasicControl; //脱开轴组，单独控制辅助轴	 
END_VAR

// Controller_3200C/Application/B0_GloabalVariables/GVL_Const
VAR_GLOBAL
	Pi			  			: LREAL := 3.1415926;	
	iCmdTypeNO		  		: INT :=50;//每种指令类型最大数量
	iTeachPtNO		  		: INT :=46;
	g_xCameraProdTrig		: BOOL;
	g_asCameraProdInfo		: ARRAY [1..gc_iMaxNrOfCameraProducts] OF L_RPP_Product;
	g_xCameraChanelComOk	: BOOL;
	g_lrLockedInfeedPos		: LREAL;
END_VAR

// Controller_3200C/Application/B0_GloabalVariables/PrgVars
VAR_GLOBAL
	(*------------------------------------------------Modbus参数设置------------------------------------------------------------*)
	ModbusServer_1							: ModbusServer;  
	//ModbusServer_2						: ModbusServer;  
	                    					
	xEnableModebus							:BOOL:=TRUE;
	tTimeOut_Modbus							:UDINT:=0;
	xReset									:BOOL;
	arOutPutData      						AT %MW0   :ARRAY[1..1700] OF INT; //示教器读写起始地址
	arInputData	   							AT %MW1800:ARRAY[1..240] OF INT;//示教器只读数据
	                                    	
	// arOutPutData2     					AT %MW2000 :ARRAY [1..1700] OF INT; //示教器读写起始地址
	// arInputData2	   						AT %MW3800:ARRAY[1..240] OF INT;//示教器只读数据
	(*------------------------------------------------Modbus参数设置------------------------------------------------------------*)
	
	(*------------------------------------------------机器人状态显示------------------------------------------------------------*)
	xSystemWarning							AT %MW1900	:BOOL;
	xSystemError							AT %MW1901	:BOOL;
	xPowerEnable							AT %MW1902	:BOOL;
	xEmergencyStop							AT %MW1903	:BOOL;
	xLED1Status	    						AT %MW1905  :BOOL;
	xLED2Status								AT %MW1906  :BOOL;
	rLED2FlashTime							:REAL;	
	LED1_TON1								:TON;	
	LED1_TON2								:TON;	
	xLock_LED1								:BOOL;	                						
	LED2_TON1								:TON;	
	LED2_TON2								:TON;	
	xLock_LED2								:BOOL;
	
	(*------------------------------------------------Infeeder编码器回零------------------------------------------------------------*)
	xSetInfeederPosition					AT %MW1130   :BOOL;	//Infeeder位置标定
	xSetOutfeederPosition					AT %MW1131   :BOOL;	//Outfeeder位置标定
	//rInfeederPosition						AT %MW1132   :REAL; //Infeeder位置显示
	//rOutfeederPosition					AT %MW1134   :REAL; //Outfeeder位置显示
	(*------------------------------------------------Infeeder编码器回零------------------------------------------------------------*)
	
	(*------------------------------------------------相机检测产品显示------------------------------------------------------------*)	
	asCameraProd_Display					 AT %MW1950 :ARRAY [1..8] OF Display_Product;  //1950+64=2014
	asBufferHandlingProd_Display			:ARRAY [1..8] OF Display_Product;  //2050+64=2114
	
	(*------------------------------------------------相机检测产品显示------------------------------------------------------------*)	
	(*------------------------------------------------机器人状态显示--------------------------------------------------------------*)	
	(*------------------------------------------------主从通信状态显示------------------------------------------------------------*)
	xMasterRobot1Status	 					AT %MW1100 :BOOL;
	xMasterRobot2Status	 					AT %MW1101 :BOOL;
	xMasterRobot3Status	 					AT %MW1102 :BOOL;
	xMasterRobot4Status	 					AT %MW1103 :BOOL;
	xMasterRobot5Status	 					AT %MW1104 :BOOL;
	xMasterRobot6Status	 					AT %MW1105 :BOOL;
	xSlaveStatus		 					AT %MW1106 :BOOL;
	xMasterCommunicationReset				AT %MW1107 :BOOL;
	xSlaveCommunicationReset    			AT %MW1108 :BOOL;
	xOutfeederStart							:BOOL;
	fb_TON_FeederStop						:TON;//关闭出料带启动信号
	xSlaveOutfeedStartSignal				:BOOL;
	xOutfeederStartHolding 					:BOOL;
	//OutfeederStartHolding					:TOF;	
	(*------------------------------------------------主从通信状态显示------------------------------------------------------------*)
	
	(*------------------------------------------------机器人自动运行------------------------------------------------------------*)
	xRunPermission							:BOOL;	                    				
	xRunOrStopPrg	    					 AT %MW800 :BOOL;  
	iCurrentPrgCmdNum						 AT %MW801 :INT:=1;  
	iCommandType							 AT %MW802 :INT;	//指令类型   
	xResetAutoRun							 AT	%MW803 :BOOL;  
	xAutoMenu		 						 AT %MW804 :BOOL;  
	ErrorID									 :UINT;	
	WarningID								 :UINT;	
	xRunInter								 AT %MW805 :BOOL;  
	xStopInter								 AT %MW806 :BOOL;	  
	iStartPrgCmdNum		 					 AT %MW807 :INT:=1; //启动程序运行行号	
	iBufferLine_HMI							 AT %MW808 :INT:=1;//缓存行
	iPickRow_HMI							 AT %MW809 :INT;
	iPickCol_HMI						 	 AT %MW810 :INT;
	iPlaceRow_HMI							 AT %MW811 :INT;
	iPlaceCol_HMI							 AT %MW812 :INT;
	
	iCommandIndex							:INT;	//指令索引
	fb_P2P									:MC_MoveDirectAbsolute;
	fb_MoveLinear							:MC_MoveLinearAbsolute;
	fb_MoveCircle							:MC_MoveCircularAbsolute;
	fb_TON									:TON;
	fb_TON2									:TON;
	t_waitime								:TIME; //ms
	xChangeMotionType						:BOOL:=TRUE;
	iAutoStep								:INT;
	xDoNextCmd								:BOOL; //
	iJumpNum								:INT; //跳转行号	
	
	//自动运行前的相机参数设置 
	rInternalTrigTime  						AT %MW820 :REAL;	//拍照周期
	rFilterTolerance_X 						AT %MW822 :REAL;	//滤波参数
	rFilterTolerance_Y 	 					AT %MW824 :REAL;
	rMinCaptureLine							AT %MW826 :REAL;	//最小抓取线
	rMaxCaptureLine							AT %MW828 :REAL;	//最大抓取线	                            	
	rMinPlaceLine							AT %MW834 :REAL;
	rMaxPlaceLine							AT %MW836 :REAL;
															//吸盘下降高度
	rSuckerDropHeight						AT %MW892 :REAL;				   		 //   3
	rBlowGasTime							AT %MW894 :REAL:=10;				   	 //   8
	rSuck_Gas_OpenTime		    			AT %MW896 :REAL:=100;				   	 //   6
	rBlow_Gas_OpenTime 						AT %MW898 :REAL;				   		 //   7
	iBox_ExceptionDeal						AT %MW870 :INT;
	iSelfadaptPickSwitch					AT %MW874 :INT;	 //节拍自适应开关		//10	
	iProdDeformation						AT %MW875 :INT;  //产品变形量			//11
	rPnPDurationNegative					:REAL;		
	rPnPDurationPositive					:REAL;
	
	rPnPDurationNegativeLimit 				AT %MW876 :REAL;	//13
	rPnPDurationPositiveLimit 				AT %MW878 :REAL;	//14
	rTorqueForwardControl					AT %MW880 :REAL:=0.7;  //转矩前馈比例系数
	                            	
	//自动运行前的皮带参数设置              	
	rProductAdd_Z							AT %MW840 :REAL;	//抓取产品高度 h
	rFollowBias_X							AT %MW842 :REAL;	//跟踪存在的静差 	//   1
	rFollowBias_Y							AT %MW844 :REAL;						//   2
	rBelt1_ClutchPra						AT %MW846 :REAL:=0.3;//跟踪时间系数     //   4
	rBelt2_ClutchPra						AT %MW848 :REAL:=0.3;					//   5
													//吸盘标定
	iSuckerNum								AT %MW850 :INT;		
	iCalibSucker							AT %MW851 :INT;
	rSuker1BiasX							AT %MW852 :REAL;
	rSuker1BiasY							AT %MW854 :REAL;
	rSuker1PickC							AT %MW1000 :REAL;
	rSuker2BiasX							AT %MW856 :REAL;
	rSuker2BiasY							AT %MW858 :REAL;
	rSuker2PickC							AT %MW1002 :REAL;
	rSuker3BiasX							AT %MW860 :REAL;
	rSuker3BiasY							AT %MW862 :REAL;
	rSuker3PickC							AT %MW1004 :REAL;
	rSuker4BiasX							AT %MW864 :REAL;
	rSuker4BiasY							AT %MW866 :REAL;
	rSuker4PickC							AT %MW1006 :REAL;
	                            			
	//标定时C轴角度   	                		
	rCalibCaxisAngle						AT %MW868 :REAL;
	xReadCalibCaxisAngle	    			AT %MW872 :BOOL;
	rBiasX									:REAL;
	rBiasY									:REAL;
	rCalibCaxisAngletoRad					:REAL;
	                            	
	//标定时C轴角度
	//rCalibCaxisAngle						AT %MW870 :REAL;	
	//xReadCalibCaxisAngle	    			AT %MW872 :BOOL;			
	//xPrgSwtich		   					AT %MW801 :BOOL:=1; //1:跟踪  2：不跟踪
	(*------------------------------------------------机器人自动运行------------------------------------------------------------*)
	                   
         	
	(*------------------------------------------------设备参数设置------------------------------------------------------------*)
	//WriteDeltaPara						:l_mc4p_writeparameter;
	WriteA1axisPara							:ARRAY[1..2] OF MC_WriteParameter;
	WriteA2axisPara							:ARRAY[1..2] OF MC_WriteParameter;
	WriteA3axisPara							:ARRAY[1..2] OF MC_WriteParameter;
	WriteAuxCaxisPara						:ARRAY[1..2] OF MC_WriteParameter;
	WriteXaxisPara							:ARRAY[1..2] OF MC_WriteParameter;
	WriteYaxisPara							:ARRAY[1..2] OF MC_WriteParameter;
	WriteZaxisPara							:ARRAY[1..2] OF MC_WriteParameter;
	//WriteInfeedPara						:MC_WriteParameter;
	//WriteOutfeedPara						:MC_WriteParameter;
	                            			
	ChangeInfeederPara  					:L_MC1P_ChangeMachineData;
	ChangeOutfeederPara						:L_MC1P_ChangeMachineData;
	InFeedPower								:MC_Power;
	OutFeedPower							:MC_Power;
	WriteA1_Step							:INT;
	WriteA2_Step							:INT;
	WriteA3_Step							:INT;
	WriteAuxC_Step							:INT;
	SetParameter_TON						:ARRAY[1..9] OF TON;//计时测算设定参数失败 
	                            	
	//初始化上载电机参数	                            	
	ReadA1axisPara							:ARRAY[1..9] OF MC_ReadParameter;
	ReadA2axisPara							:ARRAY[1..9] OF MC_ReadParameter;
	ReadA3axisPara							:ARRAY[1..9] OF MC_ReadParameter;
	ReadAuxCaxisPara						:ARRAY[1..9] OF MC_ReadParameter;
	ReadXaxisPara							:ARRAY[1..2] OF MC_ReadParameter;
	ReadYaxisPara							:ARRAY[1..2] OF MC_ReadParameter;
	ReadZaxisPara							:ARRAY[1..2] OF MC_ReadParameter;
	ReadInfeederPara  						:L_MC1P_ReadMachineData;
	ReadOutfeederPara						:L_MC1P_ReadMachineData;
	                            	
	//A1轴参数设置                   	
	rA1_PositiveLimit						AT %MW600 :REAL;
	rA1_NegativeLimit						AT %MW602 :REAL;
	rA1_Vel_P1								AT %MW604 :REAL;
	rA1_Vel_I1								AT %MW606 :REAL;
	rA1_Pos_P1								AT %MW608 :REAL;
	xA1_ConfirmPara							AT %MW614 :BOOL;
	                                		
	//A2轴参数设置                       		
	rA2_PositiveLimit						AT %MW620 :REAL;
	rA2_NegativeLimit						AT %MW622 :REAL;
	rA2_Vel_P2								AT %MW624 :REAL;
	rA2_Vel_I2								AT %MW626 :REAL;
	rA2_Pos_P2								AT %MW628 :REAL;
	xA2_ConfirmPara							AT %MW634 :BOOL;
	                            			
	//A3轴参数设置                   			
	rA3_PositiveLimit						AT %MW640 :REAL;
	rA3_NegativeLimit						AT %MW642 :REAL;
	rA3_Vel_P3								AT %MW644 :REAL;
	rA3_Vel_I3								AT %MW646 :REAL;
	rA3_Pos_P3								AT %MW648 :REAL;
	xA3_ConfirmPara							AT %MW654 :BOOL;
	
	//X轴参数设置
	rXaxis_PositiveLimit					AT %MW660 :REAL;
	rXaxis_NegativeLimit					AT %MW662 :REAL;
	xXaxis_ConfirmPara						AT %MW691 :BOOL;
	                        				
	//Y轴参数设置                				
	rYaxis_PositiveLimit					AT %MW670 :REAL;
	rYaxis_NegativeLimit					AT %MW672 :REAL;
	xYaxis_ConfirmPara						AT %MW692 :BOOL;
	                        				
	//Z轴参数设置                				
	rZaxis_PositiveLimit					AT %MW680 :REAL;
	rZaxis_NegativeLimit					AT %MW682 :REAL;
	xZaxis_ConfirmPara						AT %MW693 :BOOL;
	                                		
	//AuxC轴参数设置                     		
	rAuxC_PositiveLimit						AT %MW730 :REAL;
	rAuxC_NegativeLimit						AT %MW732 :REAL;
	rAuxC_Vel_P3							AT %MW734 :REAL;
	rAuxC_Vel_I3							AT %MW736 :REAL;
	rAuxC_Pos_P3							AT %MW738 :REAL;
	xAuxC_ConfirmPara						AT %MW740 :BOOL;
	
	//A1轴参数显示
	rA1_PositiveLimit_Dsp					AT %MW742 :REAL;
	rA1_NegativeLimit_Dsp					AT %MW744 :REAL;
	rA1_Vel_P1_Dsp							AT %MW746 :REAL;
	rA1_Vel_I1_Dsp							AT %MW748 :REAL;
	rA1_Pos_P1_Dsp							AT %MW750 :REAL;
	//A2轴参数显示                       		
	rA2_PositiveLimit_Dsp					AT %MW752 :REAL;
	rA2_NegativeLimit_Dsp					AT %MW754 :REAL;
	rA2_Vel_P1_Dsp							AT %MW756 :REAL;
	rA2_Vel_I1_Dsp							AT %MW758 :REAL;
	rA2_Pos_P1_Dsp							AT %MW760 :REAL;
	//A3轴参数显示                       		
	rA3_PositiveLimit_Dsp					AT %MW762 :REAL;
	rA3_NegativeLimit_Dsp					AT %MW764 :REAL;
	rA3_Vel_P1_Dsp							AT %MW766 :REAL;
	rA3_Vel_I1_Dsp							AT %MW768 :REAL;
	rA3_Pos_P1_Dsp							AT %MW770 :REAL;
	//AuxC轴参数显示                     		
	rAuxC_PositiveLimit_Dsp					AT %MW772 :REAL;
	rAuxC_NegativeLimit_Dsp					AT %MW774 :REAL;
	rAuxC_Vel_P1_Dsp						AT %MW776 :REAL;
	rAuxC_Vel_I1_Dsp						AT %MW778 :REAL;
	rAuxC_Pos_P1_Dsp						AT %MW780 :REAL;
	//X轴参数显示
	rXaxis_PositiveLimit_Dsp				AT %MW782 :REAL;
	rXaxis_NegativeLimit_Dsp				AT %MW784 :REAL;
	//Y轴参数显示                        		
	rYaxis_PositiveLimit_Dsp				AT %MW786 :REAL;
	rYaxis_NegativeLimit_Dsp				AT %MW788 :REAL;
	//Z轴参数显示                        		
	rZaxis_PositiveLimit_Dsp				AT %MW790 :REAL;
	rZaxis_NegativeLimit_Dsp				AT %MW792 :REAL;
	                                		
	//进料带编码器参数设置                    		
	xInfeederDirection						AT %MW900 :BOOL;//方向
	rInfeederPosResolution					AT %MW901 :REAL;//每圈线数
	rInfeederGearRedRatio					AT %MW903 :REAL;//减速比
	rInfeederFeedConst						AT %MW905 :REAL;//每圈皮带行进长度
	//rInfeederCycleLength					AT %MW907 :REAL;//皮带长度
	xInfeederConfirmParameter				AT %MW909 :BOOL;
	//进料带编码器参数显示                    		
	xInfeederDirectionDsp					AT %MW910 :BOOL;	
	rInfeederPosResolutionDsp				AT %MW911 :REAL;
	rInfeederGearRedRatioDsp				AT %MW913 :REAL;
	rInfeederFeedConstDsp					AT %MW915 :REAL;
	//rInfeederCycleLengthDsp				AT %MW917 :REAL;
	
	//出料带编码器参数设置
	xOutfeederDirection						AT %MW920 :BOOL;	//方向
	rOutfeederPosResolution					AT %MW921 :REAL;    //每圈线数
	rOutfeederGearRedRatio					AT %MW923 :REAL;    //减速比
	rOutfeederFeedConst						AT %MW925 :REAL;    //每圈皮带行进长度
	//rOutfeederCycleLength					AT %MW927 :REAL;    //皮带长度
	xOutfeederConfirmParameter				AT %MW929 :BOOL;
	
	//出料带编码器参数显示
	xOutfeederDirectionDsp					AT %MW930 :BOOL;
	rOutfeederPosResolutionDsp				AT %MW931 :REAL;
	rOutfeederGearRedRatioDsp				AT %MW933 :REAL;
	rOutfeederFeedConstDsp					AT %MW935 :REAL;
	//rOutfeederCycleLengthDsp				AT %MW937 :REAL;	
	
	//电机额定电流与实际电流
	rA1_Rated_Current						AT %MW940 :REAL;
	rA1_Actual_Current						AT %MW942 :REAL;
	rA2_Rated_Current						AT %MW944 :REAL;
	rA2_Actual_Current						AT %MW946 :REAL;
	rA3_Rated_Current						AT %MW948 :REAL;
	rA3_Actual_Current						AT %MW950 :REAL;
	rAuxC_Rated_Current						AT %MW952 :REAL;
	rAuxC_Actual_Current					AT %MW954 :REAL;
	//电机额定转矩与实际转矩               			
	rA1_Rated_Torque						AT %MW956 :REAL;
	rA1_Actual_Torque						AT %MW958 :REAL;
	rA2_Rated_Torque						AT %MW960 :REAL;
	rA2_Actual_Torque						AT %MW962 :REAL;
	rA3_Rated_Torque						AT %MW964 :REAL;
	rA3_Actual_Torque						AT %MW966 :REAL;
	rAuxC_Rated_Torque						AT %MW968 :REAL;
	rAuxC_Actual_Torque						AT %MW970 :REAL;
	                            			
	//负荷分配配置-Start	            			
	iLoadMode								AT %MW270 :INT; //负荷分配模式 NUll Master Slave
	iRobotNum								AT %MW271 :INT; //机器人数量
	iLoadProdNum							AT %MW272 :INT; //负荷分配产品数量
	iLoadDistrRule							AT %MW273 :INT; //负荷分配规则 1 密集分拣 2 平均分配
	arLoadRatio								AT %MW274 :ARRAY[1..6] OF REAL; //MW274~MW285
	aiServerCommuPort						AT %MW286 :ARRAY[1..6] OF UINT;  //MW286~MW291
	iSlaveCommuPort							AT %MW292 :UINT;	
	//负荷分配配置-End	
	(*------------------------------------------------设备参数设置------------------------------------------------------------*)
	
	(*------------------------------------------------机器人状态显示(499~550)-------------------------------------------------*)
	ReadAxis1Info							:MC_ReadAxisInfo;
	ReadAxis2Info							:MC_ReadAxisInfo;
	ReadAxis3Info							:MC_ReadAxisInfo;
	ReadAxisAuxCInfo						:MC_ReadAxisInfo;
	                        				
	iRecycleNum								:INT:=20;
	//RobotReady  							AT %MW499 :BOOL;
	RobotAxesEnable							AT %MW500 :BOOL;
	RobotAxesGroupEnable					AT %MW501 :BOOL;
	RobotHoming								AT %MW502 :BOOL;
	//RobotSWlimitEnable					AT %MW503 :BOOL;
	RobotSlimit								AT %MW504 :BOOL;
	                        	
	RobotAxesWarning						AT %MW506 :	BOOL ;
	RobotAxesError							AT %MW507 :	BOOL ;
	RobotPrgOrParaError						AT %MW505 :	BOOL ;                            
	                        				           	
	RotAxisEnable							AT %MW510 :	BOOL ;
	RotAxisHoming							AT %MW511 :	BOOL ;
	RotAxisSPlimit							AT %MW513 :	BOOL ;
	RotAxisSNlimit							AT %MW514 :	BOOL ;
	RotAxis24Warning						AT %MW517 :	BOOL ;
	RotAxisWarning							AT %MW518 :	BOOL ;
	RotAxisError							AT %MW519 :	BOOL ;
			                				           	
	A1axisEnable							AT %MW521 :	BOOL;
	A1axisHoming							AT %MW522 :	BOOL;
	A1axisSPlimit							AT %MW524 :	BOOL;
	A1axisSNlimit							AT %MW525 :	BOOL;
	A1axis24Warning							AT %MW528 :	BOOL;
	A1axisWarning							AT %MW529 : BOOL;
	A1axisError								AT %MW530 : BOOL;
						    	
	A2axisEnable		    	 			AT %MW532 :BOOL;
	A2axisHoming		    	 			AT %MW533 :BOOL;
	A2axisSPlimit		    	 			AT %MW535 :BOOL;
	A2axisSNlimit		    	 			AT %MW536 :BOOL;
	A2axis24Warning		   		 			AT %MW539 :BOOL;
	A2axisWarning		    	 			AT %MW540 :BOOL;
	A2axisError			    	 			AT %MW541 :BOOL;
						    	 			
	A3axisEnable		    	 			AT %MW543 :BOOL;
	A3axisHoming		    	 			AT %MW544 :BOOL;
	A3axisSPlimit		    	 			AT %MW546 :BOOL;
	A3axisSNlimit		    	 			AT %MW547 :BOOL;
	A3axis24Warning		    	 			AT %MW550 :BOOL;
	A3axisWarning		    	 			AT %MW551 :BOOL;
	A3axisError			    	 			AT %MW552 :BOOL;
	                        	 			
	DeltaRobot_ErrorID			 			AT %MW553 :UINT;
	Xaxis_ErrorID				 			AT %MW554 :UINT;
	Yaxis_ErrorID				 			AT %MW555 :UINT;
	Zaxis_ErrorID				 			AT %MW556 :UINT;
	                        	 			
	A1axis_ErrorID				 			AT %MW557 :UINT;
	A2axis_ErrorID				 			AT %MW558 :UINT;
	A3axis_ErrorID				 			AT %MW559 :UINT;
	AuxCaxis_ErrorID			 			AT %MW560 :UINT;
	                        	 			
	PrgOrParaErrorID			 			AT %MW561 :UINT;
	(*------------------------------------------------机器人状态显示(499~550)------------------------------------------------------------*)
	(*------------------------------------------------传送带设置------------------------------------------------------------*)
	//进料带参数
	rConveyorInRecord0						AT %MW350	:REAL;	
	rConveyorInRecord1  					AT %MW352	:REAL;	
	rConveyorInRecord2						AT %MW354	:REAL;	
	                        					
	rReadInfeedPos1_X						AT %MW356	:REAL;	
	rReadInfeedPos1_Y						AT %MW358	:REAL;	
	rReadInfeedPos1_Z						AT %MW360	:REAL;	
	                        					
	rReadInfeedPos2_X						AT %MW362	:REAL;	
	rReadInfeedPos2_Y						AT %MW364	:REAL;	
	rReadInfeedPos2_Z						AT %MW366	:REAL;	
	                        					
	rReadInfeedPos3_X						AT %MW436	:REAL;	
	rReadInfeedPos3_Y						AT %MW438	:REAL;	
	rReadInfeedPos3_Z						AT %MW440	:REAL;	
	                        			
	rReadInfeedPos4_X						AT %MW442	:REAL;	
	rReadInfeedPos4_Y						AT %MW444	:REAL;	
	rReadInfeedPos4_Z						AT %MW446	:REAL;	
	                                		    
	xInfeedRead0							AT %MW368	:BOOL;	
	xInfeedRead1							AT %MW369	:BOOL;		
	xInfeedRead2							AT %MW370	:BOOL;	
	xInfeedRead3							AT %MW448	:BOOL;		
	xInfeedRead4							AT %MW449	:BOOL;		
	                        			
	PCS5_X0									AT %MW450 	:REAL;	
	PCS5_Y0									AT %MW452 	:REAL;	
	PCS5_X1									AT %MW454 	:REAL;	
	PCS5_Y1									AT %MW456 	:REAL;	
	PCS5_X2									AT %MW458 	:REAL;	
	PCS5_Y2									AT %MW460 	:REAL;	
	PCS5_X3									AT %MW462 	:REAL;	
	PCS5_Y3									AT %MW464 	:REAL;	
	PCS5_dx									AT %MW466	:REAL;	
	PCS5_dy									AT %MW468	:REAL;	
	                        					
	PCS6_X0									AT %MW470 	:REAL;	
	PCS6_Y0									AT %MW472 	:REAL;	
	PCS6_X1									AT %MW474 	:REAL;	
	PCS6_Y1									AT %MW476 	:REAL;	
	PCS6_X2									AT %MW478 	:REAL;	
	PCS6_Y2									AT %MW480 	:REAL;	
	PCS6_X3									AT %MW482 	:REAL;	
	PCS6_Y3									AT %MW484 	:REAL;	
	PCS6_dx									AT %MW486	:REAL;	
	PCS6_dy									AT %MW488	:REAL;	
	                                			
	xCaculateInfeedBeltOrigin 				AT %MW371   :BOOL;		
	theta1									:REAL;	
	alpha									:REAL;	
	rBeta									:REAL;	
	rInfeedMapX								:REAL;	
	rInfeedMapY								:REAL;	
	rOutfeedMapX							:REAL;	
	rOutfeedMapY							:REAL;	
	//出料带参数                     			
	rConveyorOutRecord0						AT %MW380	:REAL;
	rConveyorOutRecord1  					AT %MW382	:REAL;
	rConveyorOutRecord2						AT %MW384	:REAL;
	                        				
	rReadOutfeedPos1_X						AT %MW386	:REAL;
	rReadOutfeedPos1_Y						AT %MW388	:REAL;
	rReadOutfeedPos1_Z						AT %MW390	:REAL;
	                        	    		
	rReadOutfeedPos2_X						AT %MW392	:REAL;
	rReadOutfeedPos2_Y						AT %MW394	:REAL;
	rReadOutfeedPos2_Z						AT %MW396	:REAL;
	                        				
	rReadOutfeedPos3_X						AT %MW296	:REAL;
	rReadOutfeedPos3_Y						AT %MW298	:REAL;
	rReadOutfeedPos3_Z						AT %MW300	:REAL;
	                        				
	rReadOutfeedPos4_X						AT %MW302	:REAL;
	rReadOutfeedPos4_Y						AT %MW304	:REAL;
	rReadOutfeedPos4_Z						AT %MW306	:REAL;
	                        				
	                        				
	xOutfeedRead0							AT %MW398	:BOOL;
	xOutfeedRead1							AT %MW399	:BOOL;	
	xOutfeedRead2							AT %MW400	:BOOL;	
	                        		
	xOutfeedRead3							AT %MW308	:BOOL;	
	xOutfeedRead4							AT %MW309	:BOOL;
	                            			
	xCaculateOutfeedBeltOrigin 				AT %MW401  :BOOL;	
	theta2									:REAL;
	gama									:REAL;
	//PCS5标定                        		
	PCS5_OriginX							AT %MW402 :REAL; //坐标系原点
	PCS5_OriginY							AT %MW404 :REAL;
	PCS5_OriginZ							AT %MW406 :REAL;
	PCS5_OriginA							AT %MW408 :REAL;
	PCS5_OriginB							AT %MW410 :REAL;
	PCS5_OriginC		 					AT %MW412 :REAL;
	                        		
	//PCS6标定                		
	PCS6_OriginX							AT %MW423 :REAL; //坐标系原点
	PCS6_OriginY							AT %MW425 :REAL;
	PCS6_OriginZ							AT %MW427 :REAL;
	PCS6_OriginA							AT %MW429 :REAL;
	PCS6_OriginB							AT %MW431 :REAL;
	PCS6_OriginC		 					AT %MW433 :REAL;
	                        			
	fbSetToolTransform  					:L_MC4P_SetToolTransform;
	fbSetActiveTool							:L_MC4P_SetActiveTool;
	ToolRef									:L_MC4P_TOOL_REF;
	iSetToolStep							:INT;
	fb_InfeedCalib							:L_RPP_CalBeltCalib;
	fb_OutfeedCalib							:L_RPP_CalBeltCalib;
	                                		
	fbPCS5_Calib       						:MC_SetCartesianTransform;
	fbPCS6_Calib       						:MC_SetCartesianTransform; 
	                        			
	sInFeedBeltOrigin						AT %MW1820 	:BeltOrigin;  //以上为计算进料带原点及坐标系所用数据		//1831
	sOutFeedBeltOrigin						AT %MW1880 	:BeltOrigin;	 //以上为计算出料带原点及坐标系所用数据		//1891
	xTeachRCalPt2							AT %MW372	:BOOL;
	xTeachRCalPt3							AT %MW373	:BOOL;
	xTeachRCalPt4							AT %MW374	:BOOL;
	xCaculateCameraCalPts					AT %MW375	:BOOL;
	                        				
	RobotCalPt1								AT %MW1832 :CalibratePt;	//1837
	RobotCalPt2								AT %MW1838 :CalibratePt;	//1843
	RobotCalPt3								AT %MW1844 :CalibratePt;	//1849
	RobotCalPt4								AT %MW1850 :CalibratePt;	//1855
	                        				
	CameraCalPt1							AT %MW1856 :CalibratePt;	//1861
	CameraCalPt2							AT %MW1862 :CalibratePt;	//1867
	CameraCalPt3							AT %MW1868 :CalibratePt;	//1873
	CameraCalPt4							AT %MW1874 :CalibratePt;	//1879
	
	(*------------------------------------------------传送带设置------------------------------------------------------------*)
	
	(*------------------------------------------------抱闸开关------------------------------------------------------------*)
	// Brake Open
	A1_BrakeDelay							: TOF;
	A2_BrakeDelay							: TOF;
	A3_BrakeDelay							: TOF;
	AuxC_BrakeDelay							: TOF;
	A1_BrakeControl							: L_MC1P_BrakeInterface; 
	A2_BrakeControl							: L_MC1P_BrakeInterface;
	A3_BrakeControl							: L_MC1P_BrakeInterface;
	AuxC_BrakeControl						: L_MC1P_BrakeInterface;
	fbBrakeTon								: TON;
	bA1_Open								AT %MW328 :BYTE;   //抱闸A1
	bA2_Open								AT %MW329 :BYTE;   //抱闸A2
	bA3_Open								AT %MW330 :BYTE;   //抱闸A3
	bC_Open									AT %MW331 :BYTE;   //抱闸C
	
	xA1_BrakeOpenStatus				  		:BOOL;	
	xA2_BrakeOpenStatus				  		:BOOL;	
	xA3_BrakeOpenStatus				  		:BOOL;	
	xC_BrakeOpenStatus				  		:BOOL;	
	
	bA1_BrakeOpenStatus						AT %MW332:BYTE;	
	bA2_BrakeOpenStatus						AT %MW333:BYTE;	
	bA3_BrakeOpenStatus						AT %MW334:BYTE;	
	bC_BrakeOpenStatus						AT %MW335:BYTE;	
	                                    	
	x_Suck1_HMI								AT %MW336 :BOOL;  //吸气1
	x_Blow1_HMI								AT %MW338 :BOOL;  //吹气1
	x_Suck1									:BOOL;
	x_Blow1									:BOOL;
	//g_xDoShootOut							AT %MW337 :BOOL;//相机触发开关 在GVL_HardwareIO中
	xPrgDoOutputVal							AT %MW339 :BOOL;//程序输出开关
	//xPrgDiInputVal						AT %MW344 :BOOL;//程序输入开关
	                        				
	i_Suck1_Num								AT %MW340 :INT:=5;  //吸气1 DO端口号
	i_Blow1_Num								AT %MW341 :INT:=6;  //吹气1 DO端口号
	                        				
	iDoShootOut_Num							AT %MW342 :INT:=7;  //相机触发开关 DO端口号
	iPrgDoOutputVal_Num						AT %MW343 :INT:=10;  //程序输出开关 DO端口号
	//iPrgDiInputVal_Num					AT %MW345 :INT;  //程序输入开关 DI端口号
	DO_0									AT %QX1.0:BOOL;//设备运行
	DO_1									AT %QX1.1:BOOL;//设备故障
	DO_2									AT %QX1.2:BOOL;//
	DO_3									AT %QX1.3:BOOL:=TRUE;//STO通电 松开抱闸STO关掉
	DO_4									AT %QX1.4:BOOL;
	DO_5									AT %QX1.5:BOOL;	
	DO_6									AT %QX1.6:BOOL;	
	DO_7									AT %QX1.7:BOOL;	
	
	//2017.01.09	
	(*	DO_8								AT %QX2.0:BOOL;
	DO_9									AT %QX2.1:BOOL;
	DO_10									AT %QX2.2:BOOL;
	DO_11									AT %QX2.3:BOOL;
	DO_12									AT %QX2.4:BOOL;
	DO_13									AT %QX2.5:BOOL;	
	DO_14									AT %QX2.6:BOOL;	
	DO_15									AT %QX2.7:BOOL;	*)	
	                        				
	                        				
	DI_0									AT %IX8.0:BOOL;//HMI握持信号
	DI_1									AT %IX8.1:BOOL;//手动高速
	DI_2									AT %IX8.2:BOOL;//手动低速
	DI_3									AT %IX8.3:BOOL;//检测 箱体 传感器输入
	DI_4									AT %IX8.4:BOOL;//
	DI_5									AT %IX8.5:BOOL;//对外开放
	DI_6									AT %IX8.6:BOOL;//对外开放
	DI_7									AT %IX8.7:BOOL;//对外开放
	//5、6、7作为外部等待事件接口                   	
	                                    	
	DI2_Rtrig								:R_TRIG;
	DI3_Rtrig								:R_TRIG;
	DI2_Ftrig								:F_TRIG;
	DI3_Ftrig								:F_TRIG;
	(*------------------------------------------------抱闸开关------------------------------------------------------------*)	
	xLocal_or_Remote						AT %MW300 :BOOL; //机器人本机控制 or 远程控制
	iBoxTotalPrdoNr 						AT %MW305 :INT:=72; //每箱产量
	
	(*------------------------------------------------机器人回零------------------------------------------------------------*)
	L_McSetPosition							: ARRAY[1..6] OF MC_SetPosition;
	xHomingActive							: BOOL;
	xHomingEnable							: BOOL;
	xSetA1Position							AT %MW317   :BOOL;	//A1位置标定
	xSetA2Position							AT %MW318   :BOOL;  //A2位置标定
	xSetA3Position							AT %MW319   :BOOL;	//A3位置标定
	xSetAuxCPosition						AT %MW320   :BOOL;	//AuxC位置标定
	                        				
	rA1SetHomePostion						AT %MW321	:REAL;  //A1设定零位	
	rA2SetHomePostion						AT %MW323	:REAL;  //A2设定零位
	rA3SetHomePostion						AT %MW325	:REAL;  //A3设定零位
	rAuxCSetHomePostion						AT %MW348	:REAL;  //AuxC设定零位	
	(*------------------------------------------------机器人回零------------------------------------------------------------*)	
	
	CustomerPrg								:L_RPP_CustomerProgram;//用户程序结构体包含：1、运动指令，2、索引参数，3、示教点
	CommandType								:L_RPP_CommandType;	
	i										:INT;
	j										:INT;	 
	//RdData_test							:ARRAY[1..500,1..20] OF STRING;//测试监视刷新率	
	
	(*------------------------------------------------手动、示教------------------------------------------------------------*)	
	//速度模式   		//运动模式	
	xBTtest									:BOOL; //手动按钮1
	iCurrentCS								:L_MC4P_CoordSystem;
	RobotPos		    					AT %MW1800:sRobotPos; //机器人位置显示 (只读)800+2*7-1=813  
	Robot_Vel_X								AT %MW1920:REAL;
	Robot_Vel_Y								AT %MW1922:REAL;
	Robot_Vel_Z								AT %MW1924:REAL;
	Robot_Vel_C								AT %MW1926:REAL;
	Robot_Vel_A1							AT %MW1928:REAL;
	Robot_Vel_A2							AT %MW1930:REAL;
	Robot_Vel_A3							AT %MW1932:REAL;
	Infeed_Vel								AT %MW1934:REAL;
	Outfeed_Vel								AT %MW1936:REAL;
	Infeed_Pos								AT %MW1938:REAL;
	Outfeed_Pos								AT %MW1940:REAL;
	                    					
	iCSchange								AT %MW100:INT;	//坐标系选择
	bBTMenu1								AT %MW101:BYTE; //手动按钮1 X+  A1+
	bBTMenu2								AT %MW102:BYTE; //手动按钮2	Y+  A2+
	bBTMenu3								AT %MW103:BYTE; //手动按钮3	Z+	A3+
	bBTMenu4								AT %MW104:BYTE; //手动按钮4	X-	A1-
	bBTMenu5								AT %MW105:BYTE; //手动按钮5	Y-  A2-
	bBTMenu6								AT %MW106:BYTE; //手动按钮6 Z-  A3-
	bBTMenu7								AT %MW107:BYTE; //手动按钮7 C+
	bBTMenu8								AT %MW108:BYTE; //手动按钮8 C-
	iJogVel									AT %MW109:INT :=10; //手动移动速度设置
	iSelectTeNO								AT %MW110:INT:=10; 	//选择示教点编号
	bSavePt									AT %MW111:BYTE;	 //保存当前编号示教点
	xSaveRunPra	  							AT %MW98 :BOOL;  //只保存自动运行参数
	xBox_ReadBelt							AT %MW210 :BOOL; //读取箱体在出料带原点时，出料带位置
	rBox_BeltPos							AT %MW211 :REAL; //传送带位置
	iBox_TchNo								AT %MW213 :INT:=20; // 装箱示教点编号
	xBox_Tch								AT %MW214 :BOOL; //装箱示教
	xPhoSwitch								AT %MW215 :BOOL; //光电开关检测信号输出
	rBoxLength								AT %MW216 :REAL;//箱体长度
	rBoxBiasLength							AT %MW218 :REAL;//箱体偏置长度
	iNewProdNum								AT %MW225 :INT:=1;//检测物体需要的外部触发信号数量
	rBoxOutfeederVel						AT %MW226 :REAL;// 装箱时出料带的速度
	rBoxPickTime							AT %MW228 :REAL;// 装箱抓取物料时间
	rBoxPlaceTime 							AT %MW230 :REAL;// 装箱放置物料时间
	rBoxDetectPosX							AT %MW232 :REAL;// 装箱检测箱体的初始位置
	rPallet_DeltaX							AT %MW250 :REAL;//码盘间距deltax
	rPallet_DeltaY							AT %MW252 :REAL;//码盘间距deltax
	iPrdtDetectDevice   					AT %MW220 :INT:=1;//产品检测装置选择 0：相机；1：传感器；2：上位机通讯指定
	rSensorBeltPos							AT %MW221 :REAL;//传感器相对进料带原点的位置
	rSensorAuxC								AT %MW223 :REAL;//传感器检测产品固定角度
	aLRPP_TeachPoints						AT %MW1200:ARRAY[1..50] OF L_RPP_CartesianPoint;//定义示教点	
	bCurrentPos								AT %MW1700:ARRAY[1..50] OF WORD; //获取当前机器人位置显示开关
	ReadActPos_MCS							:MC_GroupReadActualPosition;	
	ReadActPos_PCS							:MC_GroupReadActualPosition;	
	ReadActPos_ACS							:MC_GroupReadActualPosition;	
	ReadActPos_CS							:MC_GroupReadActualPosition;	
	                    					
	xTest									:BOOL; 
	axJogPos								:ARRAY[1..12] OF BOOL;
	axJogNeg								:ARRAY[1..12] OF BOOL;
	xactive_move							:BOOL;
	(*------------------------------------------------手动、示教------------------------------------------------------------*)	
	
	stCameraStartTime:              		SysTime;
	stCameraPhase1Time:             		SysTime;
	stCameraPhase2Time:             		SysTime;
	stCameraPhase3Time:             		SysTime;
	stCameraFB1Time:             			SysTime;
	stCameraFB2Time:             			SysTime;
	stCameraFB3Time:             			SysTime;	
	stCameraTotalTime:						systime;
	                                		
	stCoveyorStartTime:						systime;
	stCoveyorEndTime:						systime;
	stCoveyorWholeTime:						systime;
	                             	    	
	stMainStartTime:						systime;
	stMainEndTime:							systime;	
	stMainTotalTime:						systime;
	                                		
	stAutoRunStartTime:						systime;
	stAutoRunEndTime:						systime;	
	stAutoRunTotalTime:						systime;	
	                                		
	stCutomerPrgStartTime:					systime;
	stCutomerPrgEndTime:					systime;  
	stCutomerPrgWholeTime:					systime;  
	                                		
	stABCStartTime:							systime;
	stABCEndTime:							systime;	
	stABCTotalTime:							systime;
	                            			
	stRevStartTime:							systime;
	stRevEndTime:							systime;	
	stRevTotalTime:							systime;
END_VAR

// Controller_3200C/Application/B0_GloabalVariables/GVL_MainFlow
VAR_GLOBAL
	(*------------------------------------------------框架流程-----------------------------------------------------------*)
	//示教器不同状态切换
	//xHoming						AT %MW700:BOOL;      //1.寻零模式
	xManualMode						AT %MW701:BOOL;		 //2.手动模式
	xEditPrg						AT %MW702:BOOL;		 //3.程序编辑
	xAutoRun						AT %MW706:BOOL;		 //4.自动运行	    
	xRemoteTest				 		 :BOOL;  	//远程自动运行控制测试
	DetectRemoteControl_Trig		 :R_TRIG; //检测外部启动上升沿
	
	xJumpOutManualJog				AT %MW703 :BOOL;		
	xToolActive						AT %MW704 :BOOL;		//标定触发，激活工具坐标系
	xToolDeActive					AT %MW714 :BOOL;		//取消工具坐标系标定
	xResetError						AT %MW705 :BOOL;		//复位错误
	xTotalConfig					AT %MW707 :BOOL; 	//总配置
	iCameraType						AT %MW708 :INT; 	//相机类型选择
	xBeltCalibCSchange 				AT %MW709 :BOOL; 	//标定传送带-坐标系切换  modified in 2016 10 25
	xAuxCHome						AT %MW715 :BOOL;  	//辅助轴回零
	iHMI_InitWindow					AT %MW710 :INT;     //HMI中PLC控制元件关联变量，用以切换不同的窗口
	ChangeHMIWindow_TON  			:TON;   			//切换HMI窗口定时器
	
	xCameraHMIStatus				AT %MW716 :BOOL;		 //相机通信状态显示到HMI上
	ChangeCameraStatus_TON 			:TON;			//检测相机通信正常定时器
	DetectCameraStatus_Trig			:R_TRIG;		//检测相机通信正常触发器
	
	iWindowTest						AT %MW711 :INT;
	xInitWindow						:BOOL;
	xResetPrg						:BOOL;
	wstep							:WORD;		 	 	 //模式切换
	xMainInit	 					AT %MW712:BOOL;		 //初始化标志位
	xLogicInit						AT %MW713:BOOL;
	iInitStep						:INT;				 //初始化模式跳转
	xExternalMode					AT %MW310:BOOL;	//false：内部索引模式； true：外部索引模式 	                    			
	g_xCycleReady					:BOOL;			// 自动抓取就绪信号
	g_xCycleStop					:BOOL;			// 停止自动抓取
	g_xCycleEStop					:BOOL;			// 自动抓取紧急停止
	                    			
	g_xCameraComOk					:BOOL;
	xCameraEnable					:BOOL;		//:=TRUE;
	xSensorEnable					:BOOL;
	xComputerEnable 				:BOOL;

(*------------------------------------------------框架流程-----------------------------------------------------------*)
END_VAR

// Controller_3200C/Application/B0_GloabalVariables/PPVars
VAR_GLOBAL
	L_MC1P_AverageFilterSetValues_A1: 			L_MC1P_AverageFilterSetValues;
	L_MC1P_AverageFilterSetValues_A2: 			L_MC1P_AverageFilterSetValues;
	L_MC1P_AverageFilterSetValues_A3: 			L_MC1P_AverageFilterSetValues;
	L_MC1P_AverageFilterSetValues_A4: 			L_MC1P_AverageFilterSetValues;		
	xFilterEnable: 								BOOL:=TRUE;
	wFilterDepth: 								WORD:=30;	
	TON_0:										TON;	
END_VAR

// Controller_3200C/Application/B0_GloabalVariables/GVL_HardwareIO
VAR_GLOBAL
	g_xDoShootOut 			 AT %MW337:BOOL;//相机触发开关
	g_xReadReady			:BOOL;//相机读取完毕信号
	g_xDILockPos 			:BOOL;
	g_wEncoderControl 		:WORD:=4;   // Infeed belt Encoder
	g_wEncoderControl2 		:WORD:=4;   // Infeed belt Encoder
END_VAR

// Controller_3200C/Application/Main
PROGRAM Main
VAR
(*------------------------------------------------用户编程参数设置------------------------------------------------------------*)
(*------------------------------------------------用户编程参数设置------------------------------------------------------------*)
(*------------------------------------------------程序自动运行------------------------------------------------------------*)
(*------------------------------------------------程序自动运行------------------------------------------------------------*)
(*------------------------------------------------相机标定------------------------------------------------------------*)	
	LoadDistribution					: L_RPP_LoadDistribution;
	BufferHandling						: L_RPP_BufferHandling;	
	SensorBufferHandler					: SensorBufferhandling;
	                    				
	xSlaveBoxfull 						: BOOL;//从机箱体装满
	xMasterBoxfull  					: BOOL; //主机箱体装满
	xAllMasterLoad      				: BOOL; //主机满负载
	xAllSlaveLoad       				: BOOL; //从机满负载
	xSlaveBoxReady  					: BOOL;//从机箱体准备好
	fb_DetectAllMasterLoad 				: TON; //延时检测是否为主机完全负荷模式
	DetectSlaveBoxfull					: F_TRIG;//检测从机箱体准备信号
	
	// CameraInterface
	ipAddr								: NBS.IP_ADDR:= ( sAddr := '192.168.5.20' );
	xReStart: BOOL;	
	xAutoMode: BOOL;
	xShootInternal: BOOL;
	lrInternalTrigTime: LREAL;
	xShootTrig: BOOL;	
	//xCameraEnable	:BOOL:=TRUE;
	xFbEnable :BOOL:=TRUE;
	aTCP_Master :ARRAY[1..6] OF L_RPP_TCP_Master;	
	TCP_WriteData :L_RPP_TCP_WriteData; //专门用作主从机箱体启动信号通信-------------------2017.07.16
	axMasterEnable :ARRAY[1..6] OF BOOL;
	k	:INT;
	TCP_Slave :L_RPP_TCP_Slave;
	xSlaveEnable	:BOOL;
(*------------------------------------------------相机标定------------------------------------------------------------*)

	TransX: INT;
	TransY: INT;
	TransZ: INT;
	RotAngle1: INT;
	RotAngle2: INT;
	
//----------------------------
	xResetClearBuffer 	: BOOL;
	slrFilterTolerance	: L_RPP_Tolerance;
	ClearBuffer_Rtrig	: R_TRIG;
	Bias_X				: LREAL;
	Lock_Rtrig: R_TRIG;	
	DetectStop_Ftrig: F_TRIG;
	fb_TON_Menu		:TON;
	fb_TON_Init		:TON;	
	
	stStartTime				: SYSTIME;
	stEndTime				: SYSTIME;
	lrAxis_X_ActPosPassed,		lrAxis_Y_ActPosPassed	: LREAL;
			
	MultiPickHandling	:L_RPP_MultiPickHandling;	
	fb_TON_Delete  :TON;
	fb_TON_Delay  :TON;
	xProdInfoReady_TON: TON;
	xProductDel_TON: TON;
	xTimeFlag	:bool;
	//sFirstProdInfo: INT;
	iProd_Count		:INT;
	//**********Set Torque limit********************************************************************************
	j												: INT;
	iIntermediatePointPassed						: INT;			
	fbSetTorqueLimit								: ARRAY[1..3] OF L_MC1P_SetTorqueLimit;	
	xSetTorqueLimitEnable							: ARRAY[1..3] OF BOOL:=[TRUE,TRUE,TRUE];	
	A1_TorqueLimitFactor							: ARRAY[0..10] OF LREAL:=[ 3.0,3.0,3.0,3.0,3.0,3.0,3.0,3.0,1.0,1.0,1.0];//A1转矩限幅因数
	A2_TorqueLimitFactor							: ARRAY[0..10] OF LREAL:=[ 3.0,3.0,3.0,3.0,3.0,3.0,3.0,3.0,1.0,1.0,1.0];//A2转矩限幅因数
	A3_TorqueLimitFactor							: ARRAY[0..10] OF LREAL:=[ 3.0,3.0,3.0,3.0,3.0,3.0,3.0,3.0,1.0,1.0,1.0];//A3转矩限幅因数
	lrMotorRatedTorque								: ARRAY[1..3] OF LREAL;//A1、A2、A3电机额定转矩																						
	lrTorqueLimit									: ARRAY[1..3] OF LREAL;//A1、A2、A3 Torque Limit
			
	//*********Interface of 2 LCP_PickPlace Function Blocks**********************************************************************************************
	CoefMaxOfStartAndEndR							: ARRAY[1..2] OF LREAL:=[2,2];
	Aux1ExePointPassed								: ARRAY[1..2] OF INT:=[1,1];	
	Aux1DurationRatio								: ARRAY[1..2] OF LREAL:=[0.7,0.7];		
	Aux1MotionLaw									: ARRAY[1..2] OF INT:=[3,3];	//2: 5th ploy; 3: 7th ploy
	StartAlphaRatio									: ARRAY[1..2,1..3] OF LREAL:=[0.33,0.67,1.00, 0.30,0.67,1.00];
	EndAlphaRatio									: ARRAY[1..2,7..9] OF LREAL:=[1.00,0.67,0.25, 1.00,0.67,0.25];	
	
//************2017.03.30	
	lrDistToMinCapLForCycleAdaptive					: LREAL:=450.0;//mm
	lrMaxTimeforCycleAdaptive						: LREAL:=1.0; //s
	L_USPP_PT1Filter_0								: L_USPP_PT1Filter;
	lrInfeederFilterVelocity						: LREAL;		
	fbGroupReadActualPosition 						: MC_GroupReadActualPosition;
	fbReadCartesianTransform 						: MC_ReadCartesianTransform;
	arSetPosition_PCS								:ARRAY[1..3] OF REAL;
	RotAngle_C										:REAL;
	Tx,Ty,Tz										:REAL;
	x0,y0,z0										:REAL;
	iPlaceCounter							: INT:=0;
	fb_PlaceCounter_Triger					: R_TRIG;
	OutfeederStartOutputDelay   			: TOF;
	xDOTest									: BOOL;
	rAngle_PI								: REAL;
	rAngle									: REAL;
	rAngle2									: REAL;
	rAngle_PI2								: REAL;
	fb_TON_STO_Off							: TON;
	rAngle_a								: LREAL;
	rAngle_PI_a								: LREAL;
	rAngle_b								: LREAL;
	rAngle_PI_b								: LREAL;
	FourPts_Calibration_1 					: FourPts_Calibration; //四点标定PCS坐标系
	FourPts_Calibration_2 					: FourPts_Calibration; //四点标定PCS坐标系
	theta1,theta2							: LREAL;
//**************************************************************************************
	fb_InverseKinematics					: LCP_MC4P_InvKinOfDeltaRobot;	
	LCP_MC4P_TorqueComputation_1			: LCP_MC4P_TorqueFeedForwardControl;	
	alrCoulombFriction						: ARRAY[1..6] OF LREAL:=[3.9,3.9,3.9];
	alrViscousFriction						: ARRAY[1..6] OF LREAL:=[0.27,0.27,0.27];
	lrRatioOfTorqueFeedForward				: LREAL;
	xFeedforwardControl						: BOOL;
	xFrictionCompe							: BOOL;	
END_VAR

(*******************************外部启动自动运行界面*****************************)		

(*******************************外部启动自动运行界面***************************)
SystimeGetUs(pUsTime:= stAutoRunStartTime);	
(*******************************00——程序初始化********************************) 
		IF	NOT xMainInit  THEN			
			A00_Init();
		END_IF
(*******************************02——产品检测装置选择**************************) 
		A02_DetectDeviceChoose();		
(*******************************03——上电使能控制******************************) 
		A03_PowerCtrl();
(*******************************04——复位集成功能******************************) 	
		A04_ResetFunction();		
(*******************************20——手动控制**********************************)	
		A20_ManualJog();			
(*******************************30——自动控制**********************************)
		A30_AutoRun();		
(*******************************40——参数设置*********************************)
		A40_SetParameters();		
(*******************************80-气阀吸气吹气处理***************************)		
		A80_SuckBlow();
(*******************************91-TCP_Master*********************************)		
		
(*******************************92-TCP_Master*********************************)
		
(*******************************93——力矩限幅**********************************)	
		A93_SetTorqueLimit();
		
(*******************************外部启动自动运行界面**************************)		
	
			
(*******************************用户程序解析***************************************)		
		// 装箱参数输入
		CustomerPrgHandling.rBoxOutfeederVel:=rBoxOutfeederVel;
		CustomerPrgHandling.rBoxDetectPosX:=rBoxDetectPosX;
		CustomerPrgHandling.rBoxPickTime:=rBoxPickTime;
		CustomerPrgHandling.rBoxPlaceTime:=rBoxPlaceTime;
		//CustomerPrgHandling.rPalletDeltaX:=rPallet_DeltaX;
		//CustomerPrgHandling.rPalletDeltaY:=rPallet_DeltaY;
		
		//吸气吹气控制-放置到主进程		 modified in 2016 10 25
		x_Suck1:=CustomerPrgHandling.xSuck OR x_Suck1_HMI;
		x_Blow1:=CustomerPrgHandling.xBlow OR x_Blow1_HMI;
		
		//等待外部输入调用端口	modified in 2016 10 25
		CustomerPrgHandling.DI_5:=DI_5;
		CustomerPrgHandling.DI_6:=DI_6;
		CustomerPrgHandling.DI_7:=DI_7;

		//调用CustomerPrgHandling call 			//modified in 2016.11.03
	IF	 xMainInit  THEN							
		CustomerPrgHandling(Delta_Robot:=Delta_Robot,AuxC:=AxisYaw, Outfeeder:=Outfeeder,
		xMasterOutfeederStart:=xOutfeederStart,xSlaveOutfeederStart:=xSlaveOutfeedStartSignal,Infeeder:=Infeeder,xRunOrStopPrg:=xRunOrStopPrg,iOutputVal:=xPrgDoOutputVal,ErrorID:=ErrorID);//程序自动解析
	END_IF
(*******************************用户程序解析************************************)
	

(*******************************机器人与辅助轴非自动模式使能********************)	
	//CustomerPrgHandling.xRunPermission=false 如果CustomerPrgHandling.xRunPermission为false，则表示没有启动程序，则可以调用ABC模块

		IF NOT xAutoRun THEN//xAutoRun  
			AGBControl(AxesGroup:=Delta_Robot);//xEnableInternalControl:=TRUE
		
		END_IF
(*******************************机器人与辅助轴非自动模式使能********************)	
	
	
(*******************************如果系统错误，机器人将停止自动运行**************)
		IF xSystemError OR xEmergencyStop THEN
			xRunOrStopPrg:=FALSE;
		END_IF
(*******************************如果系统错误，机器人将停止自动运行**************)
				
(*******************************辅助轴单独控制**********************************)	
		Aux1_ABC.xEnablePositive:=TRUE;
		Aux1_ABC.xEnableNegative:=TRUE;
		Aux1_ABC.xDisableSWLimit:=FALSE;
		Aux1_ABC.xResetError:=xResetError;
		
		//辅助轴AuxC 一键回零
		IF xAuxCHome THEN
			xAuxCHome:=FALSE;
			Aux1_ABC.xMoveAbsExecute:=TRUE;
			Aux1_ABC.lrSetPos_Dist:=0;
		END_IF
		
		IF Aux1_ABC.xInPosition THEN
			Aux1_ABC.xMoveAbsExecute:=FALSE;
		END_IF
(*******************************辅助轴单独控制***********************************)	

		ChangeHMIWindow_TON();

SystimeGetUs(pUsTime:= stAutoRunEndTime);
stAutoRunTotalTime:=stAutoRunEndTime-stAutoRunStartTime;

fb_PlaceCounter_Triger(CLK:=CustomerPrgHandling.L_RPP_PickPlace_1.Done,Q=>);

A98_TFFControl();
A94_RealAxisFilter();
//A96_IK();

ACTION A00_Init:
CASE iInitStep OF
	0:
		//进料带参数
		rConveyorInRecord0:=p_rConveyorInRecord0;
		rConveyorInRecord1:=p_rConveyorInRecord1;
		rConveyorInRecord2:=p_rConveyorInRecord2;	
					
		rReadInfeedPos1_X:=p_rReadInfeedPos1_X;		
		rReadInfeedPos1_Y:=p_rReadInfeedPos1_Y;		
		rReadInfeedPos1_Z:=p_rReadInfeedPos1_Z;		
		
		rReadInfeedPos2_X:=p_rReadInfeedPos2_X;			
		rReadInfeedPos2_Y:=p_rReadInfeedPos2_Y;			
		rReadInfeedPos2_Z:=p_rReadInfeedPos2_Z;
		
		rReadInfeedPos3_X:=p_rReadInfeedPos3_X;		
		rReadInfeedPos3_Y:=p_rReadInfeedPos3_Y;		
		rReadInfeedPos3_Z:=p_rReadInfeedPos3_Z;		
		
		rReadInfeedPos4_X:=p_rReadInfeedPos4_X;			
		rReadInfeedPos4_Y:=p_rReadInfeedPos4_Y;			
		rReadInfeedPos4_Z:=p_rReadInfeedPos4_Z;
				
		theta1:=p_theta1;
		alpha:=p_alpha;
		rInfeedMapX:=p_rInfeedMapX;
		rInfeedMapY:=p_rInfeedMapY;
		
		//出料带参数
		rConveyorOutRecord0:=p_rConveyorOutRecord0;
		rConveyorOutRecord1:=p_rConveyorOutRecord1;
		rConveyorOutRecord2:=p_rConveyorOutRecord2;
		
		rReadOutfeedPos1_X:=p_rReadOutfeedPos1_X;	
		rReadOutfeedPos1_Y:=p_rReadOutfeedPos1_Y;	
		rReadOutfeedPos1_Z:=p_rReadOutfeedPos1_Z;	
							 
		rReadOutfeedPos2_X:=p_rReadOutfeedPos2_X;	
		rReadOutfeedPos2_Y:=p_rReadOutfeedPos2_Y;	
		rReadOutfeedPos2_Z:=p_rReadOutfeedPos2_Z;	
		
		rReadOutfeedPos3_X:=p_rReadOutfeedPos3_X;	
		rReadOutfeedPos3_Y:=p_rReadOutfeedPos3_Y;	
		rReadOutfeedPos3_Z:=p_rReadOutfeedPos3_Z;	
							 
		rReadOutfeedPos4_X:=p_rReadOutfeedPos4_X;	
		rReadOutfeedPos4_Y:=p_rReadOutfeedPos4_Y;	
		rReadOutfeedPos4_Z:=p_rReadOutfeedPos4_Z;	
		
		theta2:=p_theta2;			
		gama:=p_gama;	
		
		
		//PCS5标定 
		PCS5_OriginX:=p_PCS5_OriginX;		
		PCS5_OriginY:=p_PCS5_OriginY;		
		PCS5_OriginZ:=p_PCS5_OriginZ;		
		PCS5_OriginA:=p_PCS5_OriginA;		
		PCS5_OriginB:=p_PCS5_OriginB;		
		PCS5_OriginC:=p_PCS5_OriginC;		
		
		PCS5_X0:=p_PCS5_X0;
		PCS5_Y0:=p_PCS5_Y0;
		PCS5_X1:=p_PCS5_X1;
		PCS5_Y1:=p_PCS5_Y1;
		PCS5_X2:=p_PCS5_X2;
		PCS5_Y2:=p_PCS5_Y2;
		PCS5_X3:=p_PCS5_X3;
        PCS5_Y3:=p_PCS5_Y3;
	    PCS5_dx:=p_PCS5_dx;
		PCS5_dy:=p_PCS5_dy;
		
		//PCS6标定 
		PCS6_OriginX:=p_PCS6_OriginX;		
		PCS6_OriginY:=p_PCS6_OriginY;		
		PCS6_OriginZ:=p_PCS6_OriginZ;		
		PCS6_OriginA:=p_PCS6_OriginA;		
		PCS6_OriginB:=p_PCS6_OriginB;		
		PCS6_OriginC:=p_PCS6_OriginC;
		
		PCS6_X0:=p_PCS6_X0;
		PCS6_Y0:=p_PCS6_Y0;
		PCS6_X1:=p_PCS6_X1;
		PCS6_Y1:=p_PCS6_Y1;
		PCS6_X2:=p_PCS6_X2;
		PCS6_Y2:=p_PCS6_Y2;
		PCS6_X3:=p_PCS6_X3;
        PCS6_Y3:=p_PCS6_Y3;
	    PCS6_dx:=p_PCS6_dx;
		PCS6_dy:=p_PCS6_dy;	
		
		//进料带原点及坐标系
		sInFeedBeltOrigin:=p_sInFeedBeltOrigin;	
		sOutFeedBeltOrigin:=p_sOutFeedBeltOrigin;
		
		//相机标定点
		RobotCalPt1:=p_RobotCalPt1;	
		RobotCalPt2:=p_RobotCalPt2;	
		RobotCalPt3:=p_RobotCalPt3;	
		RobotCalPt4:=p_RobotCalPt4;	
		
		CameraCalPt1:=p_CameraCalPt1;
		CameraCalPt2:=p_CameraCalPt2;
		CameraCalPt3:=p_CameraCalPt3;
		CameraCalPt4:=p_CameraCalPt4;		    

   		//rCalibCaxisAngle:=p_rCalibCaxisAngle;	
		iSuckerNum:=p_iSuckerNum;
		iCalibSucker:=p_iCalibSucker;
		rSuker1BiasX:=p_rSuker1BiasX;
		rSuker1BiasY:=p_rSuker1BiasY;
		rSuker2BiasX:=p_rSuker2BiasX;
		rSuker2BiasY:=p_rSuker2BiasY;
		rSuker3BiasX:=p_rSuker3BiasX;
		rSuker3BiasY:=p_rSuker3BiasY;
		rSuker4BiasX:=p_rSuker4BiasX;
		rSuker4BiasY:=p_rSuker4BiasY;
		//装箱体初始化
		rBoxLength:=p_rBoxLength;				//箱体长度
		rBoxBiasLength:=p_rBoxBiasLength;		//箱体偏置长度//产品检测传感器初始化
		iPrdtDetectDevice:=p_iPrdtDetectDevice; //产品检测装置选择 0：相机；1：传感器；2：上位机通讯指定
		iNewProdNum:=p_iNewProdNum;
		//检测产品传感器设置
		rSensorBeltPos:=p_rSensorBeltPos;	//传感器相对进料带原点的位置
		rSensorAuxC:=p_rSensorAuxC;			//传感器检测产品固定角度                   
		iBoxTotalPrdoNr:=p_iBoxTotalPrdoNr;
		rBoxOutfeederVel:=p_rBoxOutfeederVel;// 装箱时出料带的速度
		rBoxPickTime:=p_rBoxPickTime;// 装箱抓取物料时间
		rBoxPlaceTime:=p_rBoxPlaceTime;// 装箱放置物料时间
		rBoxDetectPosX:=p_rBoxDetectPosX;// 装箱检测箱体的初始位置 
		// 负荷分配
		iLoadMode:=p_iLoadMode;
		iRobotNum:=p_iRobotNum;
		iLoadProdNum:=p_iLoadProdNum;
		iLoadDistrRule:=p_iLoadDistrRule;
		arLoadRatio:=p_arLoadRatio; 
		aiServerCommuPort:=p_aiServerCommuPort;
		iSlaveCommuPort:=p_iSlaveCommuPort;		
		
		//设置参数初始化
		rA1_PositiveLimit:=	p_rA1_PositiveLimit	;
		rA1_NegativeLimit:=	p_rA1_NegativeLimit	;
		rA1_Vel_P1		 :=	p_rA1_Vel_P1;
		rA1_Vel_I1	 	 :=	p_rA1_Vel_I1;
		rA1_Pos_P1	 	 := p_rA1_Pos_P1;	
		
		rA2_PositiveLimit:=	p_rA2_PositiveLimit	;
		rA2_NegativeLimit:=	p_rA2_NegativeLimit	;
		rA2_Vel_P2		 :=	p_rA2_Vel_P2;
		rA2_Vel_I2	 	 :=	p_rA2_Vel_I2;
		rA2_Pos_P2		 := p_rA2_Pos_P2;
		
		rA3_PositiveLimit:=	p_rA3_PositiveLimit	;
		rA3_NegativeLimit:=	p_rA3_NegativeLimit	;
		rA3_Vel_P3		 :=	p_rA3_Vel_P3;
		rA3_Vel_I3	 	 :=	p_rA3_Vel_I3;
		rA3_Pos_P3		 := p_rA3_Pos_P3;
		
		rAuxC_PositiveLimit := p_rAuxC_PositiveLimit;
		rAuxC_NegativeLimit := p_rAuxC_NegativeLimit;		
		rAuxC_Vel_P3		:= p_rAuxC_Vel_P3;	
		rAuxC_Vel_I3		:= p_rAuxC_Vel_I3;	
		rAuxC_Pos_P3		:= p_rAuxC_Pos_P3;	
		
		rXaxis_PositiveLimit:=p_rXaxis_PositiveLimit;
		rXaxis_NegativeLimit:=p_rXaxis_NegativeLimit;
		
		rYaxis_PositiveLimit:=p_rYaxis_PositiveLimit;
		rYaxis_NegativeLimit:=p_rYaxis_NegativeLimit;

		rZaxis_PositiveLimit:=p_rZaxis_PositiveLimit;
		rZaxis_NegativeLimit:=p_rZaxis_NegativeLimit;	

		xInfeederDirection		:=p_xInfeederDirection	;
		rInfeederPosResolution  :=p_rInfeederPosResolution ;
		rInfeederGearRedRatio	:=p_rInfeederGearRedRatio;
		rInfeederFeedConst	    :=p_rInfeederFeedConst;
		//rInfeederCycleLength	:=p_rInfeederCycleLength;

		xOutfeederDirection		:=p_xOutfeederDirection		;
		rOutfeederPosResolution	:=p_rOutfeederPosResolution ;
		rOutfeederGearRedRatio	:=p_rOutfeederGearRedRatio	;
		rOutfeederFeedConst		:=p_rOutfeederFeedConst		;
		//rOutfeederCycleLength	:=p_rOutfeederCycleLength	;
		
		i_Suck1_Num:=	p_i_Suck1_Num;	//吸气吹气
		i_Blow1_Num:=	p_i_Blow1_Num;	
		//iDoShootOut_Num:=p_iDoShootOut_Num;
		//iPrgDoOutputVal_Num:=p_iPrgDoOutputVal_Num;
		
		rPallet_DeltaX:=p_rPallet_DeltaX;
		rPallet_DeltaY:=p_rPallet_DeltaY;
		
		rPnPDurationNegativeLimit:=p_rPnPDurationNegativeLimit;			
		rPnPDurationPositiveLimit:=P_rPnPDurationPositiveLimit;	
		rTorqueForwardControl:=p_rTorqueForwardControl;		
		xExternalMode:=p_xExternalMode;
		
		 //机器人本机控制 or 远程控制
		fb_TON_Init.IN:=TRUE;
		fb_TON_Init.PT:=T#5S;
		
		IF fb_TON_Init.Q THEN
			iInitStep:=1;
			fb_TON_Init.IN:=FALSE;
		END_IF

	1:	//读取断电前保存的程序
		
		IF NOT xLogicInit THEN
			CustomerPrgEdit.iSaveorOpenNum:=p_iCurrentPrgNum;
			//IF p_axSavePrgNo[p_iCurrentPrgNum]=TRUE THEN
			CustomerPrgEdit.OpenPrg(axSavePrgNo:=p_axSavePrgNo,adr_iCurrentPrgNum:=p_iCurrentPrgNum,xSaveRunPra:=xSaveRunPra,
				rFollowBias_X:=rFollowBias_X,rFollowBias_Y:=rFollowBias_Y,rSuckerDropHeight:=rSuckerDropHeight,
				rBelt1_ClutchPra:=rBelt1_ClutchPra,rBelt2_ClutchPra:=rBelt2_ClutchPra,
				rSuck_Gas_OpenTime:=rSuck_Gas_OpenTime,rBlow_Gas_OpenTime:=rBlow_Gas_OpenTime,rBlowGasTime:=rBlowGasTime,
				iBox_ExceptionDeal:=iBox_ExceptionDeal,				
				iSelfadaptPickSwitch:=iSelfadaptPickSwitch,	
				rPnPDurationNegativeLimit:= rPnPDurationNegative, 
				rPnPDurationPositiveLimit:= rPnPDurationPositive, 
				iProdDeformation:=iProdDeformation,	CustomerPrg:=CustomerPrg,aLRPP_TeachPoints:=aLRPP_TeachPoints);
					
			xLogicInit:=CustomerPrgEdit.xLogicInit;		
				
			//ELSE
			//	xLogicInit:=TRUE;
			//END_IF
			
		END_IF	
	
		IF xLogicInit=TRUE THEN
			iInitStep:=2;
		END_IF
		

	2:	//设置X轴参数
		//----------启动设置失败定时器------------//
		SetParameter_TON[1].IN:=TRUE;
		SetParameter_TON[1].PT:=T#2S;
		//----------启动设置失败定时器------------//	
		WriteXaxisPara[1].Execute:=TRUE;
		WriteXaxisPara[1].ParameterNumber:=51;
		WriteXaxisPara[1].Value:=rXaxis_PositiveLimit;
		
		WriteXaxisPara[2].Execute:=TRUE;
		WriteXaxisPara[2].ParameterNumber:=52;
		WriteXaxisPara[2].Value:=rXaxis_NegativeLimit;						
		
		IF WriteXaxisPara[1].Done AND WriteXaxisPara[2].Done THEN
			FOR i:=1 TO 2 BY 1 DO
				WriteXaxisPara[i].Execute:=FALSE;
			END_FOR
			SetParameter_TON[1].IN:=FALSE;
			iInitStep:=3;
		END_IF	
		//----------设置失败复位并输出警告信息-----------//
		IF SetParameter_TON[1].Q  THEN //如果定时时间到并且设置按钮没有复位,复位并输出报警信息
				SetParameter_TON[1].IN:=FALSE;
				FOR i:=1 TO 2 BY 1 DO
					WriteXaxisPara[i].Execute:=FALSE;
				END_FOR
				//报警信息
				WarningID:=30051;
				iInitStep:=3;
		END_IF
		//----------设置失败复位并输出警告信息-----------//			
						

	3:	//设置Y轴参数
		//----------启动设置失败定时器------------//
		SetParameter_TON[2].IN:=TRUE;
		SetParameter_TON[2].PT:=T#2S;
		//----------启动设置失败定时器------------//
		WriteYaxisPara[1].Execute:=TRUE;
		WriteYaxisPara[1].ParameterNumber:=51;
		WriteYaxisPara[1].Value:=rYaxis_PositiveLimit;
		
		WriteYaxisPara[2].Execute:=TRUE;
		WriteYaxisPara[2].ParameterNumber:=52;
		WriteYaxisPara[2].Value:=rYaxis_NegativeLimit;						
		
		IF WriteYaxisPara[1].Done AND WriteYaxisPara[2].Done THEN
			FOR i:=1 TO 2 BY 1 DO
				WriteYaxisPara[i].Execute:=FALSE;
			END_FOR
			SetParameter_TON[2].IN:=FALSE;
			iInitStep:=4;
		END_IF	
		
	//----------设置失败复位并输出警告信息-----------//
		IF SetParameter_TON[2].Q  THEN //如果定时时间到并且设置按钮没有复位,复位并输出报警信息
				SetParameter_TON[2].IN:=FALSE;
				FOR i:=1 TO 2 BY 1 DO
					WriteYaxisPara[i].Execute:=FALSE;
				END_FOR
				//报警信息
				WarningID:=30052;
				iInitStep:=4;
		END_IF
	//----------设置失败复位并输出警告信息-----------//	
		
	4:	//设置Z轴参数	
		//----------启动设置失败定时器------------//
		SetParameter_TON[3].IN:=TRUE;
		SetParameter_TON[3].PT:=T#2S;
		//----------启动设置失败定时器------------//
		WriteZaxisPara[1].Execute:=TRUE;
		WriteZaxisPara[1].ParameterNumber:=51;
		WriteZaxisPara[1].Value:=rZaxis_PositiveLimit;
		
		WriteZaxisPara[2].Execute:=TRUE;
		WriteZaxisPara[2].ParameterNumber:=52;
		WriteZaxisPara[2].Value:=rZaxis_NegativeLimit;						
		
		IF WriteZaxisPara[1].Done AND WriteZaxisPara[2].Done THEN
			FOR i:=1 TO 2 BY 1 DO
				WriteZaxisPara[i].Execute:=FALSE;
			END_FOR
			SetParameter_TON[3].IN:=FALSE;
			iInitStep:=5;
		END_IF	
	//----------设置失败复位并输出警告信息-----------//
		IF SetParameter_TON[3].Q THEN //如果定时时间到并且设置按钮没有复位,复位并输出报警信息
				SetParameter_TON[3].IN:=FALSE;
				FOR i:=1 TO 2 BY 1 DO
					WriteZaxisPara[i].Execute:=FALSE;
				END_FOR
				//报警信息
				WarningID:=30053;
				iInitStep:=5;
		END_IF
	//----------设置失败复位并输出警告信息-----------//	
		
	5:	//设置A1轴参数
			//----------启动设置失败定时器------------//
			SetParameter_TON[4].IN:=TRUE;
			SetParameter_TON[4].PT:=T#2S;
			//----------启动设置失败定时器------------//
				CASE WriteA1_Step OF
				0:
					WriteA1axisPara[1].Execute:=TRUE;
					WriteA1axisPara[1].ParameterNumber:=51;
					WriteA1axisPara[1].Value:=rA1_PositiveLimit;
					IF WriteA1axisPara[1].Done THEN				
						WriteA1axisPara[1].Execute:=FALSE;
						WriteA1_Step:=1;
					END_IF
				1:
					WriteA1axisPara[1].Execute:=TRUE;
					WriteA1axisPara[1].ParameterNumber:=52;
					WriteA1axisPara[1].Value:=rA1_NegativeLimit;
					IF WriteA1axisPara[1].Done THEN				
						WriteA1axisPara[1].Execute:=FALSE;
						WriteA1_Step:=2;
					END_IF
				2:
					WriteA1axisPara[1].Execute:=TRUE;
					WriteA1axisPara[1].ParameterNumber:=L_MC1P_IndexToParameter(16#2900,1,4);
					WriteA1axisPara[1].Value:=rA1_Vel_P1*100000;
					IF WriteA1axisPara[1].Done THEN				
						WriteA1axisPara[1].Execute:=FALSE;
						WriteA1_Step:=3;
					END_IF
				3:
					WriteA1axisPara[1].Execute:=TRUE;
					WriteA1axisPara[1].ParameterNumber:=L_MC1P_IndexToParameter(16#2900,2,2);
					WriteA1axisPara[1].Value:=rA1_Vel_I1*10;
					IF WriteA1axisPara[1].Done THEN				
						WriteA1axisPara[1].Execute:=FALSE;
						WriteA1_Step:=4;
					END_IF
				
				4:
					WriteA1axisPara[1].Execute:=TRUE;
					WriteA1axisPara[1].ParameterNumber:=L_MC1P_IndexToParameter(16#2980,0,4);
					WriteA1axisPara[1].Value:=rA1_Pos_P1*100;
					IF WriteA1axisPara[1].Done THEN				
						WriteA1axisPara[1].Execute:=FALSE;
						WriteA1_Step:=0;
						SetParameter_TON[4].IN:=FALSE; //定时器复位
						iInitStep:=6;											
					END_IF
			END_CASE
			
			
	//----------设置失败复位并输出警告信息-----------//
		IF SetParameter_TON[4].Q  THEN //如果定时时间到并且设置按钮没有复位,复位并输出报警信息
				SetParameter_TON[4].IN:=FALSE;
				WriteA1axisPara[1].Execute:=FALSE;
				WriteA1_Step:=0;
				//报警信息
				WarningID:=30054;
				iInitStep:=6;
		END_IF
	//----------设置失败复位并输出警告信息-----------//				
		
	6:	//设置A2轴参数
			//----------启动设置失败定时器------------//
			SetParameter_TON[5].IN:=TRUE;
			SetParameter_TON[5].PT:=T#2S;
			//----------启动设置失败定时器------------//
			CASE WriteA2_Step OF
				0:
					WriteA2axisPara[1].Execute:=TRUE;
					WriteA2axisPara[1].ParameterNumber:=51;
					WriteA2axisPara[1].Value:=rA2_PositiveLimit;
					IF WriteA2axisPara[1].Done THEN				
						WriteA2axisPara[1].Execute:=FALSE;
						WriteA2_Step:=1;
					END_IF
				1:
					WriteA2axisPara[1].Execute:=TRUE;
					WriteA2axisPara[1].ParameterNumber:=52;
					WriteA2axisPara[1].Value:=rA2_NegativeLimit;
					IF WriteA2axisPara[1].Done THEN				
						WriteA2axisPara[1].Execute:=FALSE;
						WriteA2_Step:=2;
					END_IF
				2:
					WriteA2axisPara[1].Execute:=TRUE;
					WriteA2axisPara[1].ParameterNumber:=L_MC1P_IndexToParameter(16#3100,1,4);
					WriteA2axisPara[1].Value:=rA2_Vel_P2*100000;
					IF WriteA2axisPara[1].Done THEN				
						WriteA2axisPara[1].Execute:=FALSE;
						WriteA2_Step:=3;
					END_IF
				3:
					WriteA2axisPara[1].Execute:=TRUE;
					WriteA2axisPara[1].ParameterNumber:=L_MC1P_IndexToParameter(16#3100,2,2);
					WriteA2axisPara[1].Value:=rA2_Vel_I2*10;
					IF WriteA2axisPara[1].Done THEN				
						WriteA2axisPara[1].Execute:=FALSE;
						WriteA2_Step:=4;
					END_IF
				
				4:
					WriteA2axisPara[1].Execute:=TRUE;
					WriteA2axisPara[1].ParameterNumber:=L_MC1P_IndexToParameter(16#3180,0,4);
					WriteA2axisPara[1].Value:=rA2_Pos_P2*100;
					IF WriteA2axisPara[1].Done THEN				
						WriteA2axisPara[1].Execute:=FALSE;
						WriteA2_Step:=0;
						SetParameter_TON[5].IN:=FALSE; //定时器复位
						iInitStep:=7;
					END_IF
			END_CASE
			
	//----------设置失败复位并输出警告信息-----------//
		IF SetParameter_TON[5].Q THEN //如果定时时间到并且设置按钮没有复位,复位并输出报警信息
				SetParameter_TON[5].IN:=FALSE;
				WriteA2axisPara[1].Execute:=FALSE;
				WriteA2_Step:=0;
				//报警信息
				WarningID:=30055;
				iInitStep:=7;	
		END_IF
	//----------设置失败复位并输出警告信息-----------//			
	7:	//设置A3轴参数
			//----------启动设置失败定时器------------//
			SetParameter_TON[6].IN:=TRUE;
			SetParameter_TON[6].PT:=T#2S;
			//----------启动设置失败定时器------------//
			CASE WriteA3_Step OF
				0:
					WriteA3axisPara[1].Execute:=TRUE;
					WriteA3axisPara[1].ParameterNumber:=51;
					WriteA3axisPara[1].Value:=rA3_PositiveLimit;
					IF WriteA3axisPara[1].Done THEN				
						WriteA3axisPara[1].Execute:=FALSE;
						WriteA3_Step:=1;
					END_IF
				1:
					WriteA3axisPara[1].Execute:=TRUE;
					WriteA3axisPara[1].ParameterNumber:=52;
					WriteA3axisPara[1].Value:=rA3_NegativeLimit;
					IF WriteA3axisPara[1].Done THEN				
						WriteA3axisPara[1].Execute:=FALSE;
						WriteA3_Step:=2;
					END_IF
				2:
					WriteA3axisPara[1].Execute:=TRUE;
					WriteA3axisPara[1].ParameterNumber:=L_MC1P_IndexToParameter(16#2900,1,4);
					WriteA3axisPara[1].Value:=rA3_Vel_P3*100000;
					IF WriteA3axisPara[1].Done THEN				
						WriteA3axisPara[1].Execute:=FALSE;
						WriteA3_Step:=3;
					END_IF
				3:
					WriteA3axisPara[1].Execute:=TRUE;
					WriteA3axisPara[1].ParameterNumber:=L_MC1P_IndexToParameter(16#2900,2,2);
					WriteA3axisPara[1].Value:=rA3_Vel_I3*10;
					IF WriteA3axisPara[1].Done THEN				
						WriteA3axisPara[1].Execute:=FALSE;
						WriteA3_Step:=4;
					END_IF
				
				4:
					WriteA3axisPara[1].Execute:=TRUE;
					WriteA3axisPara[1].ParameterNumber:=L_MC1P_IndexToParameter(16#2980,0,4);
					WriteA3axisPara[1].Value:=rA3_Pos_P3*100;
					IF WriteA3axisPara[1].Done THEN				
						WriteA3axisPara[1].Execute:=FALSE;
						WriteA3_Step:=0;
						iInitStep:=8;
						SetParameter_TON[6].IN:=FALSE; //定时器复位
					END_IF
			END_CASE
			
	//----------设置失败复位并输出警告信息-----------//
		IF SetParameter_TON[6].Q  THEN //如果定时时间到并且设置按钮没有复位,复位并输出报警信息
				SetParameter_TON[6].IN:=FALSE;
				WriteA3axisPara[1].Execute:=FALSE;
				WriteA3_Step:=0;
				//报警信息
				WarningID:=30056;
				iInitStep:=8;
		END_IF
	//----------设置失败复位并输出警告信息-----------//		
	8:	
				iInitStep:=9;
			//设置AuxC轴参数
			//----------启动设置失败定时器------------//
		(*	SetParameter_TON[7].IN:=TRUE;
			SetParameter_TON[7].PT:=T#2S;
			//----------启动设置失败定时器------------//
			CASE WriteAuxC_Step OF
				0:
					WriteAuxCaxisPara[1].Execute:=TRUE;
					WriteAuxCaxisPara[1].ParameterNumber:=51;
					WriteAuxCaxisPara[1].Value:=rAuxC_PositiveLimit;
					IF WriteAuxCaxisPara[1].Done THEN				
						WriteAuxCaxisPara[1].Execute:=FALSE;
						WriteAuxC_Step:=1;
					END_IF
				1:
					WriteAuxCaxisPara[1].Execute:=TRUE;
					WriteAuxCaxisPara[1].ParameterNumber:=52;
					WriteAuxCaxisPara[1].Value:=rAuxC_NegativeLimit;
					IF WriteAuxCaxisPara[1].Done THEN				
						WriteAuxCaxisPara[1].Execute:=FALSE;
						WriteAuxC_Step:=2;
					END_IF
				2:
					WriteAuxCaxisPara[1].Execute:=TRUE;
					WriteAuxCaxisPara[1].ParameterNumber:=L_MC1P_IndexToParameter(16#3100,1,4);
					WriteAuxCaxisPara[1].Value:=rAuxC_Vel_P3*100000;
					IF WriteAuxCaxisPara[1].Done THEN				
						WriteAuxCaxisPara[1].Execute:=FALSE;
						WriteAuxC_Step:=3;
					END_IF
				3:
					WriteAuxCaxisPara[1].Execute:=TRUE;
					WriteAuxCaxisPara[1].ParameterNumber:=L_MC1P_IndexToParameter(16#3100,2,2);
					WriteAuxCaxisPara[1].Value:=rAuxC_Vel_I3*10;
					IF WriteAuxCaxisPara[1].Done THEN				
						WriteAuxCaxisPara[1].Execute:=FALSE;
						WriteAuxC_Step:=4;
					END_IF
				
				4:
					WriteAuxCaxisPara[1].Execute:=TRUE;
					WriteAuxCaxisPara[1].ParameterNumber:=L_MC1P_IndexToParameter(16#3180,0,4);
					WriteAuxCaxisPara[1].Value:=rAuxC_Pos_P3*100;
					IF WriteAuxCaxisPara[1].Done THEN				
						WriteAuxCaxisPara[1].Execute:=FALSE;
						WriteAuxC_Step:=0;
						iInitStep:=9;
						SetParameter_TON[6].IN:=FALSE; //定时器复位
					END_IF
			END_CASE
			
		
	//----------设置失败复位并输出警告信息-----------//
		IF SetParameter_TON[7].Q  THEN //如果定时时间到并且设置按钮没有复位,复位并输出报警信息
				SetParameter_TON[7].IN:=FALSE;
				WriteAuxCaxisPara[1].Execute:=FALSE;
				WriteAuxC_Step:=0;
				//报警信息
				WarningID:=30057;
				iInitStep:=9;
		END_IF *)
	//----------设置失败复位并输出警告信息-----------//	
			
	9:	
			iInitStep:=10;
			//----------启动设置失败定时器------------//
		(*	SetParameter_TON[8].IN:=TRUE;
			SetParameter_TON[8].PT:=T#2S;
			//----------启动设置失败定时器------------//	
			ChangeInfeederPara.xExecute:=TRUE;			
			ChangeInfeederPara.xOrientation:=xInfeederDirection;
			ChangeInfeederPara.xSetOrientation:=TRUE;
			
			//ChangeInfeederPara.dwPosResolution:=REAL_TO_DWORD(rInfeederPosResolution);
			//ChangeInfeederPara.xSetPosResolution:=TRUE;
			
			ChangeInfeederPara.dwGearNumerator:=REAL_TO_DWORD(rInfeederGearRedRatio*1000*rInfeederPosResolution/2048);
			ChangeInfeederPara.dwGearDenominator:=REAL_TO_DWORD(1000);	
			ChangeInfeederPara.xSetGearFactor:=TRUE;
			
			ChangeInfeederPara.lrFeedconstant:=rInfeederFeedConst;			
			ChangeInfeederPara.xSetFeedconstant:=TRUE;
			
			
			IF ChangeInfeederPara.xDone THEN
				ChangeInfeederPara.xExecute:=FALSE;
				SetParameter_TON[8].IN:=FALSE;
				iInitStep:=10;
			END_IF
	//----------设置失败复位并输出警告信息-----------//
		IF SetParameter_TON[8].Q  THEN //如果定时时间到并且设置按钮没有复位,复位并输出报警信息
				SetParameter_TON[8].IN:=FALSE;
				ChangeInfeederPara.xExecute:=FALSE;
				//报警信息
				WarningID:=30058;
				iInitStep:=10;
		END_IF *)
	//----------设置失败复位并输出警告信息-----------//
	10:	
			iInitStep:=11;
			//----------启动设置失败定时器------------//
			(*SetParameter_TON[9].IN:=TRUE;
			SetParameter_TON[9].PT:=T#2S;
			//----------启动设置失败定时器------------//	
			ChangeOutfeederPara.xExecute:=TRUE;
			
			ChangeOutfeederPara.xOrientation:=xOutfeederDirection;
			ChangeOutfeederPara.xSetOrientation:=TRUE;
			
			//ChangeOutfeederPara.dwPosResolution:=REAL_TO_DWORD(rOutfeederPosResolution);
			//ChangeOutfeederPara.xSetPosResolution:=TRUE;
			
			ChangeOutfeederPara.dwGearNumerator:=REAL_TO_DWORD(rOutfeederGearRedRatio*1000*rOutfeederPosResolution/2048);
			ChangeOutfeederPara.dwGearDenominator:=REAL_TO_DWORD(1000);	
			ChangeOutfeederPara.xSetGearFactor:=TRUE;
			
			ChangeOutfeederPara.lrFeedconstant:=rOutfeederFeedConst;			
			ChangeOutfeederPara.xSetFeedconstant:=TRUE;
			
			//ChangeOutfeederPara.lrCycleLength:=rOutfeederCycleLength;
			//ChangeOutfeederPara.xSetCycleLength:=TRUE;
			
			IF ChangeOutfeederPara.xDone THEN
				ChangeOutfeederPara.xExecute:=FALSE;
				SetParameter_TON[9].IN:=FALSE;
				iInitStep:=11;
			END_IF
		//----------设置失败复位并输出警告信息-----------//
		IF SetParameter_TON[9].Q THEN //如果定时时间到并且设置按钮没有复位,复位并输出报警信息
				SetParameter_TON[9].IN:=FALSE;
				ChangeOutfeederPara.xExecute:=FALSE;
				//报警信息
				WarningID:=30059;
				iInitStep:=11;
		END_IF
	//----------设置失败复位并输出警告信息-----------//	*)
			
	11:	//进料带出料带标定
		fbPCS5_Calib.TransX:=p_sInFeedBeltOrigin.rOriginPosX;
		fbPCS5_Calib.TransY:=p_sInFeedBeltOrigin.rOriginPosY;
		fbPCS5_Calib.TransZ:=p_sInFeedBeltOrigin.rOriginPosZ;
		fbPCS5_Calib.RotAngle1:=p_sInFeedBeltOrigin.rRotation_A;
		fbPCS5_Calib.RotAngle2:=p_sInFeedBeltOrigin.rRotation_B;
		fbPCS5_Calib.RotAngle3:=p_sInFeedBeltOrigin.rRotation_C;
		fbPCS5_Calib.Execute:=TRUE;
		fbPCS5_Calib.CoordSystem:=L_MC4P_CoordSystem.PCS_5;
		
		fbPCS6_Calib.TransX:=p_sOutFeedBeltOrigin.rOriginPosX;
		fbPCS6_Calib.TransY:=p_sOutFeedBeltOrigin.rOriginPosY;
		fbPCS6_Calib.TransZ:=p_sOutFeedBeltOrigin.rOriginPosZ;
		fbPCS6_Calib.RotAngle1:=p_sOutFeedBeltOrigin.rRotation_A;
		fbPCS6_Calib.RotAngle2:=p_sOutFeedBeltOrigin.rRotation_B;
		fbPCS6_Calib.RotAngle3:=p_sOutFeedBeltOrigin.rRotation_C;
		fbPCS6_Calib.Execute:=TRUE;
		fbPCS6_Calib.CoordSystem:=L_MC4P_CoordSystem.PCS_6;		
		
		IF fbPCS5_Calib.Done=TRUE AND fbPCS6_Calib.Done=TRUE THEN
			fbPCS5_Calib.Execute:=FALSE;
			fbPCS6_Calib.Execute:=FALSE;
			iInitStep:=12;
		END_IF
	12:
		iInitStep:=0;
		xMainInit:=TRUE;
END_CASE
	
	fbPCS5_Calib(AxesGroup:=Delta_Robot);
	fbPCS6_Calib(AxesGroup:=Delta_Robot);
	
	fb_TON_Init();
END_ACTION

ACTION A20_ManualJog:
IF NOT xAutoRun  AND xMainInit THEN	
	
	//手动运动快捷键速度调整
		IF DI_1 THEN
			iJogVel:=100;//乘以系数0.1
		END_IF
		IF DI_2 THEN
			iJogVel:=1;//乘以系数0.1
		END_IF
		IF NOT DI_1 AND NOT DI_2 THEN
			iJogVel:=10;//10;//乘以系数0.1
		END_IF
	//手动运动快捷键速度调整



	//1. 状态变为Stangby		
	xManualMode:=FALSE;	

	//2. 手动速度设置
	AGBControl.scPar.lrCartesianJogVel:=iJogVel;   //X Y Z 
	AGBControl.scPar.lrOrientationJogVel:=iJogVel; // A B C
	AGBControl.scPar.lrRealAxisJogVel:=iJogVel*0.5;    // A1 A2 A3 C
	//modified in 2016.11.03
	Aux1_ABC.lrJoggingSetVel:=iJogVel;
	
	//3. Jog运动  //modified in 2016.11.03
	IF AGBControl.eAxesGroupState=L_MC4P_AxesGroup_State.GroupStandby AND Aux1_ABC.eFunStateAct=L_MC1P_ABC_State.Standby THEN	
							xactive_move:=TRUE;
	END_IF
	
	IF xactive_move (*AND DI_0 *) THEN	
		IF DI_0 THEN
			axJogPos[1]:=BYTE_TO_BOOL(bBTMenu1);
			axJogPos[2]:=BYTE_TO_BOOL(bBTMenu2);
			axJogPos[3]:=BYTE_TO_BOOL(bBTMenu3);
		(*	IF AGBControl.eCoordSystem=L_MC4P_CoordSystem.ACS THEN
				axJogPos[7]:=BYTE_TO_BOOL(bBTMenu7);
				ELSE
				axJogPos[7]:=BYTE_TO_BOOL(bBTMenu7);	
			END_IF *)
			Aux1_ABC.xJoggingPos:=BYTE_TO_BOOL(bBTMenu7);	//modified in 2016.11.03
						
			axJogNeg[1]:=BYTE_TO_BOOL(bBTMenu4);
			axJogNeg[2]:=BYTE_TO_BOOL(bBTMenu5);
			axJogNeg[3]:=BYTE_TO_BOOL(bBTMenu6);
			(*IF AGBControl.eCoordSystem=L_MC4P_CoordSystem.ACS THEN
				axJogNeg[7]:=BYTE_TO_BOOL(bBTMenu8);
			ELSE
				axJogNeg[7]:=BYTE_TO_BOOL(bBTMenu8);
			END_IF *)
			Aux1_ABC.xJoggingNeg:=BYTE_TO_BOOL(bBTMenu8);
			
		ELSIF NOT DI_0 THEN
			axJogPos[1]:=FALSE;
			axJogPos[2]:=false;
			axJogPos[3]:=FALSE;
			axJogPos[4]:=FALSE;
			axJogPos[6]:=FALSE;
			axJogNeg[7]:=FALSE;
			
			axJogNeg[1]:=FALSE;
			axJogNeg[2]:=FALSE;
			axJogNeg[3]:=FALSE;
			axJogPos[4]:=FALSE;
			axJogNeg[6]:=FALSE;
			axJogNeg[7]:=FALSE;
			Aux1_ABC.xJoggingPos:=FALSE;
			Aux1_ABC.xJoggingNeg:=FALSE;
		END_IF
	END_IF
	
	IF xBeltCalibCSchange THEN  // modified in 2016 10 25
		xBeltCalibCSchange:=FALSE;
		icschange:=0;	
	END_IF	
	
